LIN {X 0,Y 54.725,Z 1004.951,A -85,B 0,C 180,E1 26696.4,E2 26696.4} C_VEL
LIN {X 0,Y 49.29,Z 1006.172,A -85,B 0,C 180,E1 26729.997,E2 26729.997} C_VEL
LIN {X 0,Y 55.176,Z 1004.813,A -85,B 0,C 180,E1 26764.669,E2 26764.669} C_VEL
LIN {X 0,Y 77.211,Z 999.62,A -85,B 0,C 180,E1 26791.14,E2 26791.14} C_VEL
LIN {X 0,Y 112.41,Z 988.546,A -85,B 0,C 180,E1 26806.899,E2 26806.899} C_VEL
LIN {X 0,Y 149.803,Z 972.339,A -85,B 0,C 180,E1 26814.847,E2 26814.847} C_VEL
LIN {X 0,Y 181.716,Z 954.19,A -85,B 0,C 180,E1 26818.987,E2 26818.987} C_VEL
LIN {X 0,Y 144.346,Z 975.766,A -85,B 0,C 180,E1 26823.995,E2 26823.995} C_VEL
LIN {X 0,Y 128.492,Z 982.899,A -85,B 0,C 180,E1 26825.01,E2 26825.01} C_VEL
LIN {X 0,Y 112.377,Z 989.197,A -85,B 0,C 180,E1 26826.364,E2 26826.364} C_VEL
LIN {X 0,Y 79.371,Z 1000.218,A -85,B 0,C 180,E1 26837.491,E2 26837.491} C_VEL
LIN {X 0,Y 55.922,Z 1006.134,A -85,B 0,C 180,E1 26855.689,E2 26855.689} C_VEL
LIN {X 0,Y 42.006,Z 1009.143,A -85,B 0,C 180,E1 26888.877,E2 26888.877} C_VEL
LIN {X 0,Y 41.08,Z 1009.561,A -85,B 0,C 180,E1 26910.004,E2 26910.004} C_VEL
LIN {X 0,Y 47.227,Z 1008.017,A -85,B 0,C 180,E1 26949.886,E2 26949.886} C_VEL
LIN {X 0,Y 72.99,Z 1001.942,A -85,B 0,C 180,E1 26978.989,E2 26978.989} C_VEL
LIN {X 0,Y 110.548,Z 989.976,A -85,B 0,C 180,E1 26993.218,E2 26993.218} C_VEL
LIN {X 0,Y 149.583,Z 972.768,A -85,B 0,C 180,E1 26999.986,E2 26999.986} C_VEL
LIN {X 0,Y 157.146,Z 968.791,A -85,B 0,C 180,E1 27000.897,E2 27000.897} C_VEL
LIN {X 0,Y 117.393,Z 986.578,A -85,B 0,C 180,E1 27007.391,E2 27007.391} C_VEL
LIN {X 0,Y 80.336,Z 998.373,A -85,B 0,C 180,E1 27019.545,E2 27019.545} C_VEL
LIN {X 0,Y 57.052,Z 1003.65,A -85,B 0,C 180,E1 27037.231,E2 27037.231} C_VEL
LIN {X 0,Y 42.679,Z 1006.187,A -85,B 0,C 180,E1 27069.217,E2 27069.217} C_VEL
LIN {X 0,Y 41.362,Z 1006.47,A -85,B 0,C 180,E1 27089.996,E2 27089.996} C_VEL
LIN {X 0,Y 48.252,Z 1005.227,A -85,B 0,C 180,E1 27128.867,E2 27128.867} C_VEL
LIN {X 0,Y 74.683,Z 999.672,A -85,B 0,C 180,E1 27157.32,E2 27157.32} C_VEL
LIN {X 0,Y 107.56,Z 990.05,A -85,B 0,C 180,E1 27170.175,E2 27170.175} C_VEL
LIN {X 0,Y 148.509,Z 973.045,A -85,B 0,C 180,E1 27177.848,E2 27177.848} C_VEL
LIN {X 0,Y 157.303,Z 968.587,A -85,B 0,C 180,E1 27179.047,E2 27179.047} C_VEL
LIN {X 0,Y 117.818,Z 987.13,A -85,B 0,C 180,E1 27185.169,E2 27185.169} C_VEL
LIN {X 0,Y 112.377,Z 989.197,A -85,B 0,C 180,E1 27186.364,E2 27186.364} C_VEL
LIN {X 0,Y 96.022,Z 994.659,A -85,B 0,C 180,E1 27188.194,E2 27188.194} C_VEL
LIN {X 0,Y 79.547,Z 999.256,A -85,B 0,C 180,E1 27190.754,E2 27190.754} C_VEL
LIN {X 0,Y 51.572,Z 1005.826,A -85,B 0,C 180,E1 27208.272,E2 27208.272} C_VEL
LIN {X 0,Y 34.624,Z 1008.841,A -85,B 0,C 180,E1 27244.074,E2 27244.074} C_VEL
LIN {X 0,Y 33.124,Z 1009.263,A -85,B 0,C 180,E1 27270.005,E2 27270.005} C_VEL
LIN {X 0,Y 41.332,Z 1007.713,A -85,B 0,C 180,E1 27317.114,E2 27317.114} C_VEL
LIN {X 0,Y 70.453,Z 1001.634,A -85,B 0,C 180,E1 27345.266,E2 27345.266} C_VEL
LIN {X 0,Y 109.878,Z 989.667,A -85,B 0,C 180,E1 27357.503,E2 27357.503} C_VEL
LIN {X 0,Y 130.15,Z 981.612,A -85,B 0,C 180,E1 27361.203,E2 27361.203} C_VEL
LIN {X 0,Y 90.059,Z 995.489,A -85,B 0,C 180,E1 27369.654,E2 27369.654} C_VEL
LIN {X 0,Y 52.552,Z 1003.953,A -85,B 0,C 180,E1 27390.187,E2 27390.187} C_VEL
LIN {X 0,Y 35.329,Z 1006.487,A -85,B 0,C 180,E1 27424.618,E2 27424.618} C_VEL
LIN {X 0,Y 33.432,Z 1006.767,A -85,B 0,C 180,E1 27449.995,E2 27449.995} C_VEL
LIN {X 0,Y 42.315,Z 1005.527,A -85,B 0,C 180,E1 27495.689,E2 27495.689} C_VEL
LIN {X 0,Y 71.254,Z 1000.131,A -85,B 0,C 180,E1 27522.975,E2 27522.975} C_VEL
LIN {X 0,Y 106.472,Z 990.358,A -85,B 0,C 180,E1 27534.505,E2 27534.505} C_VEL
LIN {X 0,Y 130.541,Z 981.353,A -85,B 0,C 180,E1 27538.734,E2 27538.734} C_VEL
LIN {X 0,Y 97.059,Z 994.001,A -85,B 0,C 180,E1 27545.348,E2 27545.348} C_VEL
LIN {X 0,Y 79.547,Z 999.256,A -85,B 0,C 180,E1 27550.754,E2 27550.754} C_VEL
LIN {X 0,Y 63.154,Z 1003.048,A -85,B 0,C 180,E1 27554.617,E2 27554.617} C_VEL
LIN {X 0,Y 46.807,Z 1005.725,A -85,B 0,C 180,E1 27560.829,E2 27560.829} C_VEL
LIN {X 0,Y 27.615,Z 1008.539,A -85,B 0,C 180,E1 27596.758,E2 27596.758} C_VEL
LIN {X 0,Y 25.173,Z 1008.965,A -85,B 0,C 180,E1 27630.007,E2 27630.007} C_VEL
LIN {X 0,Y 36.292,Z 1007.408,A -85,B 0,C 180,E1 27686.561,E2 27686.561} C_VEL
LIN {X 0,Y 68.821,Z 1001.325,A -85,B 0,C 180,E1 27711.915,E2 27711.915} C_VEL
LIN {X 0,Y 98.808,Z 993.077,A -85,B 0,C 180,E1 27719.979,E2 27719.979} C_VEL
LIN {X 0,Y 103.722,Z 991.501,A -85,B 0,C 180,E1 27721.403,E2 27721.403} C_VEL
LIN {X 0,Y 60.756,Z 1002.242,A -85,B 0,C 180,E1 27734.393,E2 27734.393} C_VEL
LIN {X 0,Y 37.143,Z 1005.853,A -85,B 0,C 180,E1 27755.379,E2 27755.379} C_VEL
LIN {X 0,Y 25.522,Z 1007.064,A -85,B 0,C 180,E1 27809.994,E2 27809.994} C_VEL
LIN {X 0,Y 37.141,Z 1005.83,A -85,B 0,C 180,E1 27864.611,E2 27864.611} C_VEL
LIN {X 0,Y 69.31,Z 1000.437,A -85,B 0,C 180,E1 27889.418,E2 27889.418} C_VEL
LIN {X 0,Y 104.061,Z 991.318,A -85,B 0,C 180,E1 27898.558,E2 27898.558} C_VEL
LIN {X 0,Y 79.726,Z 998.59,A -85,B 0,C 180,E1 27904.443,E2 27904.443} C_VEL
LIN {X 0,Y 46.807,Z 1005.725,A -85,B 0,C 180,E1 27920.829,E2 27920.829} C_VEL
LIN {X 0,Y 31.263,Z 1007.541,A -85,B 0,C 180,E1 27932.406,E2 27932.406} C_VEL
LIN {X 0,Y 18.242,Z 1008.423,A -85,B 0,C 180,E1 27961.128,E2 27961.128} C_VEL
LIN {X 0,Y 17.205,Z 1008.666,A -85,B 0,C 180,E1 27990.01,E2 27990.01} C_VEL
LIN {X 0,Y 32.535,Z 1007.104,A -85,B 0,C 180,E1 28058.563,E2 28058.563} C_VEL
LIN {X 0,Y 72.688,Z 1000.024,A -85,B 0,C 180,E1 28079.971,E2 28079.971} C_VEL
LIN {X 0,Y 75.712,Z 999.346,A -85,B 0,C 180,E1 28080.652,E2 28080.652} C_VEL
LIN {X 0,Y 75.747,Z 999.286,A -85,B 0,C 180,E1 28081.86,E2 28081.86} C_VEL
LIN {X 0,Y 46.564,Z 1004.559,A -85,B 0,C 180,E1 28092.699,E2 28092.699} C_VEL
LIN {X 0,Y 21.994,Z 1007.085,A -85,B 0,C 180,E1 28126.485,E2 28126.485} C_VEL
LIN {X 0,Y 17.586,Z 1007.361,A -85,B 0,C 180,E1 28169.991,E2 28169.991} C_VEL
LIN {X 0,Y 33.143,Z 1006.131,A -85,B 0,C 180,E1 28236.005,E2 28236.005} C_VEL
LIN {X 0,Y 71.832,Z 1000.033,A -85,B 0,C 180,E1 28257.107,E2 28257.107} C_VEL
LIN {X 0,Y 75.745,Z 999.224,A -85,B 0,C 180,E1 28258.051,E2 28258.051} C_VEL
LIN {X 0,Y 75.707,Z 999.286,A -85,B 0,C 180,E1 28259.309,E2 28259.309} C_VEL
LIN {X 0,Y 42.748,Z 1005.659,A -85,B 0,C 180,E1 28272.114,E2 28272.114} C_VEL
LIN {X 0,Y 18.242,Z 1008.423,A -85,B 0,C 180,E1 28321.128,E2 28321.128} C_VEL
LIN {X 0,Y 13.954,Z 1008.54,A -85,B 0,C 180,E1 28348.35,E2 28348.35} C_VEL
LIN {X 0,Y 15.046,Z 1008,A -85,B 0,C 180,E1 28411.087,E2 28411.087} C_VEL
LIN {X 0,Y 45.426,Z 1004.937,A -85,B 0,C 180,E1 28440.165,E2 28440.165} C_VEL
LIN {X 0,Y 45.476,Z 1004.862,A -85,B 0,C 180,E1 28442.695,E2 28442.695} C_VEL
LIN {X 0,Y 17.115,Z 1007.384,A -85,B 0,C 180,E1 28467.769,E2 28467.769} C_VEL
LIN {X 0,Y 9.672,Z 1007.658,A -85,B 0,C 180,E1 28529.983,E2 28529.983} C_VEL
LIN {X 0,Y 30.76,Z 1006.434,A -85,B 0,C 180,E1 28609.855,E2 28609.855} C_VEL
LIN {X 0,Y 48.958,Z 1004.307,A -85,B 0,C 180,E1 28618.648,E2 28618.648} C_VEL
LIN {X 0,Y 16.67,Z 1007.934,A -85,B 0,C 180,E1 28644.759,E2 28644.759} C_VEL
LIN {X 0,Y 9.233,Z 1008.367,A -85,B 0,C 180,E1 28710.018,E2 28710.018} C_VEL
LIN {X 0,Y 15.046,Z 1008,A -85,B 0,C 180,E1 28771.087,E2 28771.087} C_VEL
LIN {X 0,Y 13.156,Z 1007.91,A -85,B 0,C 180,E1 28781.084,E2 28781.084} C_VEL
LIN {X 0,Y 3.411,Z 1007.913,A -85,B 0,C 180,E1 28817.533,E2 28817.533} C_VEL
LIN {X 0,Y 1.73,Z 1007.956,A -85,B 0,C 180,E1 28889.904,E2 28889.904} C_VEL
LIN {X 0,Y 8.337,Z 1007.838,A -85,B 0,C 180,E1 28980.252,E2 28980.252} C_VEL
LIN {X 0,Y 1.252,Z 1008.068,A -85,B 0,C 180,E1 29070.132,E2 29070.132} C_VEL
LIN {X 0,Y 8.174,Z 1007.847,A -85,B 0,C 180,E1 29159.743,E2 29159.743} C_VEL
LIN {X 0,Y 3.411,Z 1007.913,A -85,B 0,C 180,E1 29177.533,E2 29177.533} C_VEL
LIN {X 0,Y 1.959,Z 1009.913,A -85,B 0,C 180,E1 29207.521,E2 29207.521} C_VEL
LIN {X 0,Y 1.959,Z 1028,A -85,B 0,C 180,E1 29207.521,E2 29207.521} C_VEL
LIN {X 0,Y 1.959,Z 1028,A -85,B 0,C 180,E1 29207.521,E2 29207.521}

QRS_NEXT_CUT()
PTP {E1 29336.836,E2 29336.836}
PTP {X 0,Y 607.909,A -85,B 0,C 180,E1 29336.836,E2 29336.836,E3 0,E4 0,E5 0,E6 0}
QRS_SPEED_INIT()
LIN {X 0,Y 607.909,Z 1028,A -85,B 0,C 180,E1 29336.836,E2 29336.836,E3 0,E4 0,E5 0,E6 0} C_VEL
LIN {X 0,Y 607.909,Z 365.402,A -85,B 0,C 180,E1 29336.836,E2 29336.836} C_VEL
LIN {X 0,Y 607.909,Z 357.325,A -85,B 0,C 180,E1 29336.836,E2 29336.836} C_VEL
LIN {X 0,Y 607.881,Z 355.325,A -85,B 0,C 180,E1 29336.648,E2 29336.648} C_VEL
LIN {X 0,Y 607.838,Z 355.326,A -85,B 0,C 180,E1 29333.767,E2 29333.767} C_VEL
LIN {X 0,Y 607.91,Z 355.324,A -85,B 0,C 180,E1 29330.656,E2 29330.656} C_VEL
LIN {X 0,Y 607.845,Z 355.325,A -85,B 0,C 180,E1 29327.652,E2 29327.652} C_VEL
LIN {X 0,Y 607.919,Z 355.322,A -85,B 0,C 180,E1 29324.513,E2 29324.513} C_VEL
LIN {X 0,Y 607.851,Z 355.324,A -85,B 0,C 180,E1 29321.49,E2 29321.49} C_VEL
LIN {X 0,Y 607.914,Z 355.322,A -85,B 0,C 180,E1 29318.382,E2 29318.382} C_VEL
LIN {X 0,Y 607.857,Z 355.323,A -85,B 0,C 180,E1 29315.304,E2 29315.304} C_VEL
LIN {X 0,Y 607.917,Z 355.32,A -85,B 0,C 180,E1 29312.153,E2 29312.153} C_VEL
LIN {X 0,Y 607.865,Z 355.323,A -85,B 0,C 180,E1 29309.123,E2 29309.123} C_VEL
LIN {X 0,Y 607.915,Z 355.319,A -85,B 0,C 180,E1 29305.98,E2 29305.98} C_VEL
LIN {X 0,Y 607.873,Z 355.324,A -85,B 0,C 180,E1 29302.867,E2 29302.867} C_VEL
LIN {X 0,Y 607.914,Z 355.318,A -85,B 0,C 180,E1 29299.607,E2 29299.607} C_VEL
LIN {X 0,Y 607.902,Z 355.326,A -85,B 0,C 180,E1 29296.353,E2 29296.353} C_VEL
LIN {X 0,Y 607.886,Z 355.318,A -85,B 0,C 180,E1 29293.089,E2 29293.089} C_VEL
LIN {X 0,Y 607.913,Z 355.327,A -85,B 0,C 180,E1 29289.964,E2 29289.964} C_VEL
LIN {X 0,Y 607.907,Z 355.443,A -85,B 0,C 180,E1 29287.748,E2 29287.748} C_VEL
LIN {X 0,Y 607.908,Z 361.77,A -85,B 0,C 180,E1 29287.31,E2 29287.31} C_VEL
LIN {X 0,Y 607.919,Z 569.3,A -85,B 0,C 180,E1 29284.345,E2 29284.345} C_VEL
LIN {X 0,Y 607.911,Z 708.358,A -85,B 0,C 180,E1 29282.392,E2 29282.392} C_VEL
LIN {X 0,Y 607.914,Z 731.612,A -85,B 0,C 180,E1 29281.897,E2 29281.897} C_VEL
LIN {X 0,Y 607.916,Z 750.464,A -85,B 0,C 180,E1 29281.352,E2 29281.352} C_VEL
LIN {X 0,Y 607.912,Z 771.604,A -85,B 0,C 180,E1 29280.596,E2 29280.596} C_VEL
LIN {X 0,Y 607.917,Z 792.337,A -85,B 0,C 180,E1 29279.67,E2 29279.67} C_VEL
LIN {X 0,Y 607.916,Z 812.983,A -85,B 0,C 180,E1 29278.591,E2 29278.591} C_VEL
LIN {X 0,Y 607.917,Z 832.838,A -85,B 0,C 180,E1 29277.358,E2 29277.358} C_VEL
LIN {X 0,Y 607.912,Z 852.097,A -85,B 0,C 180,E1 29275.993,E2 29275.993} C_VEL
LIN {X 0,Y 607.909,Z 870.534,A -85,B 0,C 180,E1 29274.483,E2 29274.483} C_VEL
LIN {X 0,Y 607.916,Z 888.688,A -85,B 0,C 180,E1 29272.786,E2 29272.786} C_VEL
LIN {X 0,Y 607.914,Z 904.514,A -85,B 0,C 180,E1 29271.109,E2 29271.109} C_VEL
LIN {X 0,Y 607.913,Z 919.726,A -85,B 0,C 180,E1 29269.251,E2 29269.251} C_VEL
LIN {X 0,Y 607.913,Z 934.238,A -85,B 0,C 180,E1 29267.218,E2 29267.218} C_VEL
LIN {X 0,Y 607.896,Z 945.78,A -85,B 0,C 180,E1 29265.354,E2 29265.354} C_VEL
LIN {X 0,Y 607.887,Z 956.548,A -85,B 0,C 180,E1 29263.311,E2 29263.311} C_VEL
LIN {X 0,Y 607.91,Z 965.19,A -85,B 0,C 180,E1 29261.382,E2 29261.382} C_VEL
LIN {X 0,Y 607.892,Z 972.898,A -85,B 0,C 180,E1 29259.275,E2 29259.275} C_VEL
LIN {X 0,Y 607.89,Z 978.472,A -85,B 0,C 180,E1 29257.37,E2 29257.37} C_VEL
LIN {X 0,Y 607.909,Z 983.246,A -85,B 0,C 180,E1 29255.189,E2 29255.189} C_VEL
LIN {X 0,Y 607.882,Z 986.013,A -85,B 0,C 180,E1 29253.3,E2 29253.3} C_VEL
LIN {X 0,Y 607.909,Z 987.728,A -85,B 0,C 180,E1 29251.131,E2 29251.131} C_VEL
LIN {X 0,Y 607.883,Z 987.816,A -85,B 0,C 180,E1 29249.152,E2 29249.152} C_VEL
LIN {X 0,Y 607.886,Z 986.458,A -85,B 0,C 180,E1 29246.983,E2 29246.983} C_VEL
LIN {X 0,Y 607.904,Z 983.715,A -85,B 0,C 180,E1 29244.999,E2 29244.999} C_VEL
LIN {X 0,Y 607.88,Z 979.476,A -85,B 0,C 180,E1 29242.914,E2 29242.914} C_VEL
LIN {X 0,Y 607.914,Z 973.793,A -85,B 0,C 180,E1 29240.916,E2 29240.916} C_VEL
LIN {X 0,Y 607.889,Z 966.368,A -85,B 0,C 180,E1 29238.81,E2 29238.81} C_VEL
LIN {X 0,Y 607.89,Z 957.44,A -85,B 0,C 180,E1 29236.785,E2 29236.785} C_VEL
LIN {X 0,Y 607.911,Z 947.433,A -85,B 0,C 180,E1 29234.842,E2 29234.842} C_VEL
LIN {X 0,Y 607.904,Z 935.365,A -85,B 0,C 180,E1 29232.864,E2 29232.864} C_VEL
LIN {X 0,Y 607.903,Z 922.36,A -85,B 0,C 180,E1 29230.996,E2 29230.996} C_VEL
LIN {X 0,Y 607.913,Z 907.831,A -85,B 0,C 180,E1 29229.193,E2 29229.193} C_VEL
LIN {X 0,Y 607.915,Z 890.666,A -85,B 0,C 180,E1 29227.324,E2 29227.324} C_VEL
LIN {X 0,Y 607.905,Z 873.391,A -85,B 0,C 180,E1 29225.671,E2 29225.671} C_VEL
LIN {X 0,Y 607.908,Z 855.212,A -85,B 0,C 180,E1 29224.163,E2 29224.163} C_VEL
LIN {X 0,Y 607.914,Z 834.209,A -85,B 0,C 180,E1 29222.643,E2 29222.643} C_VEL
LIN {X 0,Y 607.917,Z 814.952,A -85,B 0,C 180,E1 29221.436,E2 29221.436} C_VEL
LIN {X 0,Y 607.918,Z 794.18,A -85,B 0,C 180,E1 29220.33,E2 29220.33} C_VEL
LIN {X 0,Y 607.914,Z 774.981,A -85,B 0,C 180,E1 29219.458,E2 29219.458} C_VEL
LIN {X 0,Y 607.913,Z 753.274,A -85,B 0,C 180,E1 29218.648,E2 29218.648} C_VEL
LIN {X 0,Y 607.911,Z 734.978,A -85,B 0,C 180,E1 29218.103,E2 29218.103} C_VEL
LIN {X 0,Y 607.912,Z 713.659,A -85,B 0,C 180,E1 29217.607,E2 29217.607} C_VEL
LIN {X 0,Y 607.916,Z 678.046,A -85,B 0,C 180,E1 29217.076,E2 29217.076} C_VEL
LIN {X 0,Y 607.907,Z 467.252,A -85,B 0,C 180,E1 29214.12,E2 29214.12} C_VEL
LIN {X 0,Y 607.908,Z 361.202,A -85,B 0,C 180,E1 29212.58,E2 29212.58} C_VEL
LIN {X 0,Y 607.905,Z 355.327,A -85,B 0,C 180,E1 29212.137,E2 29212.137} C_VEL
LIN {X 0,Y 607.891,Z 355.32,A -85,B 0,C 180,E1 29208.989,E2 29208.989} C_VEL
LIN {X 0,Y 607.916,Z 355.327,A -85,B 0,C 180,E1 29205.79,E2 29205.79} C_VEL
LIN {X 0,Y 607.907,Z 355.318,A -85,B 0,C 180,E1 29202.532,E2 29202.532} C_VEL
LIN {X 0,Y 607.887,Z 355.324,A -85,B 0,C 180,E1 29199.291,E2 29199.291} C_VEL
LIN {X 0,Y 607.915,Z 355.318,A -85,B 0,C 180,E1 29196.15,E2 29196.15} C_VEL
LIN {X 0,Y 607.874,Z 355.324,A -85,B 0,C 180,E1 29192.987,E2 29192.987} C_VEL
LIN {X 0,Y 607.915,Z 355.32,A -85,B 0,C 180,E1 29189.891,E2 29189.891} C_VEL
LIN {X 0,Y 607.866,Z 355.324,A -85,B 0,C 180,E1 29186.739,E2 29186.739} C_VEL
LIN {X 0,Y 607.916,Z 355.321,A -85,B 0,C 180,E1 29183.65,E2 29183.65} C_VEL
LIN {X 0,Y 607.858,Z 355.324,A -85,B 0,C 180,E1 29180.51,E2 29180.51} C_VEL
LIN {X 0,Y 607.917,Z 355.323,A -85,B 0,C 180,E1 29177.418,E2 29177.418} C_VEL
LIN {X 0,Y 607.851,Z 355.324,A -85,B 0,C 180,E1 29174.363,E2 29174.363} C_VEL
LIN {X 0,Y 607.918,Z 355.323,A -85,B 0,C 180,E1 29171.287,E2 29171.287} C_VEL
LIN {X 0,Y 607.845,Z 355.325,A -85,B 0,C 180,E1 29168.228,E2 29168.228} C_VEL
LIN {X 0,Y 607.911,Z 355.324,A -85,B 0,C 180,E1 29165.19,E2 29165.19} C_VEL
LIN {X 0,Y 607.837,Z 355.326,A -85,B 0,C 180,E1 29162.074,E2 29162.074} C_VEL
LIN {X 0,Y 607.89,Z 355.325,A -85,B 0,C 180,E1 29159.152,E2 29159.152} C_VEL
LIN {X 0,Y 607.832,Z 355.327,A -85,B 0,C 180,E1 29156.039,E2 29156.039} C_VEL
LIN {X 0,Y 607.846,Z 355.327,A -85,B 0,C 180,E1 29153.293,E2 29153.293} C_VEL
LIN {X 0,Y 607.837,Z 355.327,A -85,B 0,C 180,E1 29150.054,E2 29150.054} C_VEL
LIN {X 0,Y 607.833,Z 355.327,A -85,B 0,C 180,E1 29147.363,E2 29147.363} C_VEL
LIN {X 0,Y 607.874,Z 355.325,A -85,B 0,C 180,E1 29144.181,E2 29144.181} C_VEL
LIN {X 0,Y 607.837,Z 355.326,A -85,B 0,C 180,E1 29141.291,E2 29141.291} C_VEL
LIN {X 0,Y 607.904,Z 355.323,A -85,B 0,C 180,E1 29138.179,E2 29138.179} C_VEL
LIN {X 0,Y 607.842,Z 355.325,A -85,B 0,C 180,E1 29135.2,E2 29135.2} C_VEL
LIN {X 0,Y 607.919,Z 355.323,A -85,B 0,C 180,E1 29132.154,E2 29132.154} C_VEL
LIN {X 0,Y 607.85,Z 355.324,A -85,B 0,C 180,E1 29129.122,E2 29129.122} C_VEL
LIN {X 0,Y 607.918,Z 355.325,A -85,B 0,C 180,E1 29126.113,E2 29126.113} C_VEL
LIN {X 0,Y 607.857,Z 355.324,A -85,B 0,C 180,E1 29122.985,E2 29122.985} C_VEL
LIN {X 0,Y 607.915,Z 355.323,A -85,B 0,C 180,E1 29119.882,E2 29119.882} C_VEL
LIN {X 0,Y 607.863,Z 355.323,A -85,B 0,C 180,E1 29116.769,E2 29116.769} C_VEL
LIN {X 0,Y 607.913,Z 355.323,A -85,B 0,C 180,E1 29113.687,E2 29113.687} C_VEL
LIN {X 0,Y 607.869,Z 355.324,A -85,B 0,C 180,E1 29110.639,E2 29110.639} C_VEL
LIN {X 0,Y 607.914,Z 355.567,A -85,B 0,C 180,E1 29109.746,E2 29109.746} C_VEL
LIN {X 0,Y 607.913,Z 391.305,A -85,B 0,C 180,E1 29107.362,E2 29107.362} C_VEL
LIN {X 0,Y 607.916,Z 598.672,A -85,B 0,C 180,E1 29104.399,E2 29104.399} C_VEL
LIN {X 0,Y 607.913,Z 738.085,A -85,B 0,C 180,E1 29102.441,E2 29102.441} C_VEL
LIN {X 0,Y 607.915,Z 761.196,A -85,B 0,C 180,E1 29101.953,E2 29101.953} C_VEL
LIN {X 0,Y 607.916,Z 780.557,A -85,B 0,C 180,E1 29101.394,E2 29101.394} C_VEL
LIN {X 0,Y 607.911,Z 802.013,A -85,B 0,C 180,E1 29100.624,E2 29100.624} C_VEL
LIN {X 0,Y 607.919,Z 822.106,A -85,B 0,C 180,E1 29099.726,E2 29099.726} C_VEL
LIN {X 0,Y 607.916,Z 842.821,A -85,B 0,C 180,E1 29098.645,E2 29098.645} C_VEL
LIN {X 0,Y 607.916,Z 862.611,A -85,B 0,C 180,E1 29097.418,E2 29097.418} C_VEL
LIN {X 0,Y 607.912,Z 881.995,A -85,B 0,C 180,E1 29096.046,E2 29096.046} C_VEL
LIN {X 0,Y 607.91,Z 900.18,A -85,B 0,C 180,E1 29094.558,E2 29094.558} C_VEL
LIN {X 0,Y 607.916,Z 918.622,A -85,B 0,C 180,E1 29092.837,E2 29092.837} C_VEL
LIN {X 0,Y 607.91,Z 934.895,A -85,B 0,C 180,E1 29091.11,E2 29091.11} C_VEL
LIN {X 0,Y 607.91,Z 950.072,A -85,B 0,C 180,E1 29089.252,E2 29089.252} C_VEL
LIN {X 0,Y 607.911,Z 964.528,A -85,B 0,C 180,E1 29087.219,E2 29087.219} C_VEL
LIN {X 0,Y 607.9,Z 976.044,A -85,B 0,C 180,E1 29085.354,E2 29085.354} C_VEL
LIN {X 0,Y 607.886,Z 986.76,A -85,B 0,C 180,E1 29083.312,E2 29083.312} C_VEL
LIN {X 0,Y 607.907,Z 995.299,A -85,B 0,C 180,E1 29081.401,E2 29081.401} C_VEL
LIN {X 0,Y 607.896,Z 1003.04,A -85,B 0,C 180,E1 29079.275,E2 29079.275} C_VEL
LIN {X 0,Y 607.888,Z 1008.591,A -85,B 0,C 180,E1 29077.37,E2 29077.37} C_VEL
LIN {X 0,Y 607.911,Z 1013.32,A -85,B 0,C 180,E1 29075.19,E2 29075.19} C_VEL
LIN {X 0,Y 607.881,Z 1016.139,A -85,B 0,C 180,E1 29073.239,E2 29073.239} C_VEL
LIN {X 0,Y 607.897,Z 1017.761,A -85,B 0,C 180,E1 29071.037,E2 29071.037} C_VEL
LIN {X 0,Y 607.886,Z 1017.806,A -85,B 0,C 180,E1 29069.152,E2 29069.152} C_VEL
LIN {X 0,Y 607.884,Z 1016.405,A -85,B 0,C 180,E1 29066.984,E2 29066.984} C_VEL
LIN {X 0,Y 607.907,Z 1013.64,A -85,B 0,C 180,E1 29065,E2 29065} C_VEL
LIN {X 0,Y 607.882,Z 1009.103,A -85,B 0,C 180,E1 29062.82,E2 29062.82} C_VEL
LIN {X 0,Y 607.904,Z 1003.346,A -85,B 0,C 180,E1 29060.821,E2 29060.821} C_VEL
LIN {X 0,Y 607.898,Z 995.791,A -85,B 0,C 180,E1 29058.714,E2 29058.714} C_VEL
LIN {X 0,Y 607.888,Z 987.227,A -85,B 0,C 180,E1 29056.786,E2 29056.786} C_VEL
LIN {X 0,Y 607.911,Z 977.193,A -85,B 0,C 180,E1 29054.842,E2 29054.842} C_VEL
LIN {X 0,Y 607.908,Z 965.052,A -85,B 0,C 180,E1 29052.861,E2 29052.861} C_VEL
LIN {X 0,Y 607.906,Z 951.236,A -85,B 0,C 180,E1 29050.897,E2 29050.897} C_VEL
LIN {X 0,Y 607.91,Z 936.603,A -85,B 0,C 180,E1 29049.092,E2 29049.092} C_VEL
LIN {X 0,Y 607.914,Z 920.209,A -85,B 0,C 180,E1 29047.323,E2 29047.323} C_VEL
LIN {X 0,Y 607.905,Z 902.853,A -85,B 0,C 180,E1 29045.67,E2 29045.67} C_VEL
LIN {X 0,Y 607.908,Z 884.65,A -85,B 0,C 180,E1 29044.164,E2 29044.164} C_VEL
LIN {X 0,Y 607.913,Z 864.224,A -85,B 0,C 180,E1 29042.689,E2 29042.689} C_VEL
LIN {X 0,Y 607.916,Z 844.862,A -85,B 0,C 180,E1 29041.476,E2 29041.476} C_VEL
LIN {X 0,Y 607.918,Z 824.383,A -85,B 0,C 180,E1 29040.384,E2 29040.384} C_VEL
LIN {X 0,Y 607.914,Z 805.451,A -85,B 0,C 180,E1 29039.523,E2 29039.523} C_VEL
LIN {X 0,Y 607.914,Z 783.164,A -85,B 0,C 180,E1 29038.69,E2 29038.69} C_VEL
LIN {X 0,Y 607.913,Z 764.563,A -85,B 0,C 180,E1 29038.137,E2 29038.137} C_VEL
LIN {X 0,Y 607.912,Z 742.819,A -85,B 0,C 180,E1 29037.636,E2 29037.636} C_VEL
LIN {X 0,Y 607.915,Z 700.755,A -85,B 0,C 180,E1 29037.02,E2 29037.02} C_VEL
LIN {X 0,Y 607.904,Z 492.11,A -85,B 0,C 180,E1 29034.092,E2 29034.092} C_VEL
LIN {X 0,Y 607.913,Z 390.704,A -85,B 0,C 180,E1 29032.619,E2 29032.619} C_VEL
LIN {X 0,Y 607.914,Z 355.327,A -85,B 0,C 180,E1 29030.229,E2 29030.229} C_VEL
LIN {X 0,Y 607.867,Z 355.323,A -85,B 0,C 180,E1 29027.189,E2 29027.189} C_VEL
LIN {X 0,Y 607.917,Z 355.326,A -85,B 0,C 180,E1 29024.056,E2 29024.056} C_VEL
LIN {X 0,Y 607.864,Z 355.323,A -85,B 0,C 180,E1 29020.983,E2 29020.983} C_VEL
LIN {X 0,Y 607.913,Z 355.328,A -85,B 0,C 180,E1 29017.842,E2 29017.842} C_VEL
LIN {X 0,Y 607.857,Z 355.323,A -85,B 0,C 180,E1 29014.804,E2 29014.804} C_VEL
LIN {X 0,Y 607.908,Z 355.327,A -85,B 0,C 180,E1 29011.646,E2 29011.646} C_VEL
LIN {X 0,Y 607.849,Z 355.323,A -85,B 0,C 180,E1 29008.706,E2 29008.706} C_VEL
LIN {X 0,Y 607.919,Z 355.327,A -85,B 0,C 180,E1 29005.63,E2 29005.63} C_VEL
LIN {X 0,Y 607.841,Z 355.325,A -85,B 0,C 180,E1 29002.638,E2 29002.638} C_VEL
LIN {X 0,Y 607.916,Z 355.326,A -85,B 0,C 180,E1 28999.556,E2 28999.556} C_VEL
LIN {X 0,Y 607.835,Z 355.326,A -85,B 0,C 180,E1 28996.533,E2 28996.533} C_VEL
LIN {X 0,Y 607.894,Z 355.326,A -85,B 0,C 180,E1 28993.602,E2 28993.602} C_VEL
LIN {X 0,Y 607.831,Z 355.327,A -85,B 0,C 180,E1 28990.52,E2 28990.52} C_VEL
LIN {X 0,Y 607.857,Z 355.327,A -85,B 0,C 180,E1 28987.656,E2 28987.656} C_VEL
LIN {X 0,Y 607.837,Z 355.327,A -85,B 0,C 180,E1 28984.528,E2 28984.528} C_VEL
LIN {X 0,Y 607.836,Z 355.327,A -85,B 0,C 180,E1 28981.791,E2 28981.791} C_VEL
LIN {X 0,Y 607.865,Z 355.325,A -85,B 0,C 180,E1 28978.586,E2 28978.586} C_VEL
LIN {X 0,Y 607.881,Z 355.325,A -85,B 0,C 180,E1 28976.648,E2 28976.648} C_VEL
LIN {X 0,Y 606.822,Z 355.456,A -85,B 0,C 180,E1 28975.922,E2 28975.922} C_VEL
LIN {X 0,Y 600.411,Z 356.253,A -85,B 0,C 180,E1 28973.885,E2 28973.885} C_VEL
LIN {X 0,Y 599.924,Z 356.316,A -85,B 0,C 180,E1 28973.355,E2 28973.355} C_VEL
LIN {X 0,Y 599.914,Z 356.314,A -85,B 0,C 180,E1 28970.115,E2 28970.115} C_VEL
LIN {X 0,Y 599.922,Z 356.315,A -85,B 0,C 180,E1 28967.291,E2 28967.291} C_VEL
LIN {X 0,Y 599.927,Z 356.311,A -85,B 0,C 180,E1 28964.038,E2 28964.038} C_VEL
LIN {X 0,Y 599.928,Z 356.313,A -85,B 0,C 180,E1 28961.136,E2 28961.136} C_VEL
LIN {X 0,Y 599.934,Z 356.31,A -85,B 0,C 180,E1 28957.873,E2 28957.873} C_VEL
LIN {X 0,Y 599.945,Z 356.313,A -85,B 0,C 180,E1 28954.851,E2 28954.851} C_VEL
LIN {X 0,Y 599.934,Z 356.31,A -85,B 0,C 180,E1 28951.626,E2 28951.626} C_VEL
LIN {X 0,Y 599.965,Z 356.315,A -85,B 0,C 180,E1 28948.557,E2 28948.557} C_VEL
LIN {X 0,Y 599.933,Z 356.308,A -85,B 0,C 180,E1 28945.367,E2 28945.367} C_VEL
LIN {X 0,Y 599.978,Z 356.315,A -85,B 0,C 180,E1 28942.294,E2 28942.294} C_VEL
LIN {X 0,Y 599.936,Z 356.311,A -85,B 0,C 180,E1 28939.082,E2 28939.082} C_VEL
LIN {X 0,Y 599.971,Z 356.313,A -85,B 0,C 180,E1 28935.904,E2 28935.904} C_VEL
LIN {X 0,Y 599.939,Z 356.308,A -85,B 0,C 180,E1 28932.835,E2 28932.835} C_VEL
LIN {X 0,Y 599.97,Z 356.315,A -85,B 0,C 180,E1 28929.782,E2 28929.782} C_VEL
LIN {X 0,Y 599.967,Z 356.378,A -85,B 0,C 180,E1 28928.269,E2 28928.269} C_VEL
LIN {X 0,Y 601.089,Z 359.961,A -85,B 0,C 180,E1 28927.92,E2 28927.92} C_VEL
LIN {X 0,Y 601.275,Z 362.256,A -85,B 0,C 180,E1 28927.787,E2 28927.787} C_VEL
LIN {X 0,Y 601.536,Z 366.664,A -85,B 0,C 180,E1 28927.702,E2 28927.702} C_VEL
LIN {X 0,Y 601.303,Z 574.213,A -85,B 0,C 180,E1 28924.708,E2 28924.708} C_VEL
LIN {X 0,Y 601.145,Z 709.258,A -85,B 0,C 180,E1 28922.788,E2 28922.788} C_VEL
LIN {X 0,Y 601.066,Z 733.04,A -85,B 0,C 180,E1 28922.266,E2 28922.266} C_VEL
LIN {X 0,Y 601,Z 752.537,A -85,B 0,C 180,E1 28921.688,E2 28921.688} C_VEL
LIN {X 0,Y 600.875,Z 775.465,A -85,B 0,C 180,E1 28920.827,E2 28920.827} C_VEL
LIN {X 0,Y 600.791,Z 794.591,A -85,B 0,C 180,E1 28919.948,E2 28919.948} C_VEL
LIN {X 0,Y 600.649,Z 816.578,A -85,B 0,C 180,E1 28918.752,E2 28918.752} C_VEL
LIN {X 0,Y 600.552,Z 835.962,A -85,B 0,C 180,E1 28917.513,E2 28917.513} C_VEL
LIN {X 0,Y 600.414,Z 856.076,A -85,B 0,C 180,E1 28916.024,E2 28916.024} C_VEL
LIN {X 0,Y 600.306,Z 874.696,A -85,B 0,C 180,E1 28914.447,E2 28914.447} C_VEL
LIN {X 0,Y 600.224,Z 891.736,A -85,B 0,C 180,E1 28912.784,E2 28912.784} C_VEL
LIN {X 0,Y 600.132,Z 907.933,A -85,B 0,C 180,E1 28910.987,E2 28910.987} C_VEL
LIN {X 0,Y 600.07,Z 922.642,A -85,B 0,C 180,E1 28909.134,E2 28909.134} C_VEL
LIN {X 0,Y 600.012,Z 936.173,A -85,B 0,C 180,E1 28907.152,E2 28907.152} C_VEL
LIN {X 0,Y 599.975,Z 948.523,A -85,B 0,C 180,E1 28905.066,E2 28905.066} C_VEL
LIN {X 0,Y 599.926,Z 957.943,A -85,B 0,C 180,E1 28903.197,E2 28903.197} C_VEL
LIN {X 0,Y 599.911,Z 966.752,A -85,B 0,C 180,E1 28901.146,E2 28901.146} C_VEL
LIN {X 0,Y 599.914,Z 973.815,A -85,B 0,C 180,E1 28899.109,E2 28899.109} C_VEL
LIN {X 0,Y 599.884,Z 979.713,A -85,B 0,C 180,E1 28896.988,E2 28896.988} C_VEL
LIN {X 0,Y 599.904,Z 983.883,A -85,B 0,C 180,E1 28894.875,E2 28894.875} C_VEL
LIN {X 0,Y 599.896,Z 986.682,A -85,B 0,C 180,E1 28892.77,E2 28892.77} C_VEL
LIN {X 0,Y 599.885,Z 987.84,A -85,B 0,C 180,E1 28890.668,E2 28890.668} C_VEL
LIN {X 0,Y 599.913,Z 987.679,A -85,B 0,C 180,E1 28888.567,E2 28888.567} C_VEL
LIN {X 0,Y 599.888,Z 985.894,A -85,B 0,C 180,E1 28886.465,E2 28886.465} C_VEL
LIN {X 0,Y 599.9,Z 982.918,A -85,B 0,C 180,E1 28884.453,E2 28884.453} C_VEL
LIN {X 0,Y 599.917,Z 977.946,A -85,B 0,C 180,E1 28882.242,E2 28882.242} C_VEL
LIN {X 0,Y 599.893,Z 971.963,A -85,B 0,C 180,E1 28880.213,E2 28880.213} C_VEL
LIN {X 0,Y 599.929,Z 963.811,A -85,B 0,C 180,E1 28878.045,E2 28878.045} C_VEL
LIN {X 0,Y 599.957,Z 954.654,A -85,B 0,C 180,E1 28876.017,E2 28876.017} C_VEL
LIN {X 0,Y 599.969,Z 943.986,A -85,B 0,C 180,E1 28874.041,E2 28874.041} C_VEL
LIN {X 0,Y 600.019,Z 931.599,A -85,B 0,C 180,E1 28872.046,E2 28872.046} C_VEL
LIN {X 0,Y 600.075,Z 917.688,A -85,B 0,C 180,E1 28870.131,E2 28870.131} C_VEL
LIN {X 0,Y 600.16,Z 901.624,A -85,B 0,C 180,E1 28868.193,E2 28868.193} C_VEL
LIN {X 0,Y 600.254,Z 885.004,A -85,B 0,C 180,E1 28866.439,E2 28866.439} C_VEL
LIN {X 0,Y 600.349,Z 867.341,A -85,B 0,C 180,E1 28864.819,E2 28864.819} C_VEL
LIN {X 0,Y 600.476,Z 847.548,A -85,B 0,C 180,E1 28863.228,E2 28863.228} C_VEL
LIN {X 0,Y 600.576,Z 828.468,A -85,B 0,C 180,E1 28861.894,E2 28861.894} C_VEL
LIN {X 0,Y 600.716,Z 807.691,A -85,B 0,C 180,E1 28860.651,E2 28860.651} C_VEL
LIN {X 0,Y 600.81,Z 787.451,A -85,B 0,C 180,E1 28859.612,E2 28859.612} C_VEL
LIN {X 0,Y 600.94,Z 765.942,A -85,B 0,C 180,E1 28858.703,E2 28858.703} C_VEL
LIN {X 0,Y 601.012,Z 746.205,A -85,B 0,C 180,E1 28858.017,E2 28858.017} C_VEL
LIN {X 0,Y 601.11,Z 723.027,A -85,B 0,C 180,E1 28857.4,E2 28857.4} C_VEL
LIN {X 0,Y 601.155,Z 703.845,A -85,B 0,C 180,E1 28857.033,E2 28857.033} C_VEL
LIN {X 0,Y 601.392,Z 482.167,A -85,B 0,C 180,E1 28853.887,E2 28853.887} C_VEL
LIN {X 0,Y 601.358,Z 362.629,A -85,B 0,C 180,E1 28852.135,E2 28852.135} C_VEL
LIN {X 0,Y 601.083,Z 360.672,A -85,B 0,C 180,E1 28852.042,E2 28852.042} C_VEL
LIN {X 0,Y 600.876,Z 359.126,A -85,B 0,C 180,E1 28851.913,E2 28851.913} C_VEL
LIN {X 0,Y 599.958,Z 356.317,A -85,B 0,C 180,E1 28851.631,E2 28851.631} C_VEL
LIN {X 0,Y 599.971,Z 356.309,A -85,B 0,C 180,E1 28848.44,E2 28848.44} C_VEL
LIN {X 0,Y 599.944,Z 356.313,A -85,B 0,C 180,E1 28845.232,E2 28845.232} C_VEL
LIN {X 0,Y 599.97,Z 356.311,A -85,B 0,C 180,E1 28842.062,E2 28842.062} C_VEL
LIN {X 0,Y 599.938,Z 356.309,A -85,B 0,C 180,E1 28838.902,E2 28838.902} C_VEL
LIN {X 0,Y 599.976,Z 356.315,A -85,B 0,C 180,E1 28835.681,E2 28835.681} C_VEL
LIN {X 0,Y 599.94,Z 356.31,A -85,B 0,C 180,E1 28832.52,E2 28832.52} C_VEL
LIN {X 0,Y 599.955,Z 356.314,A -85,B 0,C 180,E1 28829.229,E2 28829.229} C_VEL
LIN {X 0,Y 599.954,Z 356.309,A -85,B 0,C 180,E1 28826.081,E2 28826.081} C_VEL
LIN {X 0,Y 599.93,Z 356.313,A -85,B 0,C 180,E1 28822.847,E2 28822.847} C_VEL
LIN {X 0,Y 599.963,Z 356.31,A -85,B 0,C 180,E1 28819.774,E2 28819.774} C_VEL
LIN {X 0,Y 599.921,Z 356.312,A -85,B 0,C 180,E1 28816.621,E2 28816.621} C_VEL
LIN {X 0,Y 599.96,Z 356.311,A -85,B 0,C 180,E1 28813.591,E2 28813.591} C_VEL
LIN {X 0,Y 599.915,Z 356.315,A -85,B 0,C 180,E1 28810.467,E2 28810.467} C_VEL
LIN {X 0,Y 599.936,Z 356.312,A -85,B 0,C 180,E1 28807.566,E2 28807.566} C_VEL
LIN {X 0,Y 599.912,Z 356.315,A -85,B 0,C 180,E1 28804.397,E2 28804.397} C_VEL
LIN {X 0,Y 599.917,Z 356.314,A -85,B 0,C 180,E1 28801.528,E2 28801.528} C_VEL
LIN {X 0,Y 599.908,Z 356.315,A -85,B 0,C 180,E1 28798.281,E2 28798.281} C_VEL
LIN {X 0,Y 599.899,Z 356.316,A -85,B 0,C 180,E1 28795.507,E2 28795.507} C_VEL
LIN {X 0,Y 599.91,Z 356.316,A -85,B 0,C 180,E1 28792.242,E2 28792.242} C_VEL
LIN {X 0,Y 599.891,Z 356.316,A -85,B 0,C 180,E1 28789.436,E2 28789.436} C_VEL
LIN {X 0,Y 599.94,Z 356.315,A -85,B 0,C 180,E1 28786.293,E2 28786.293} C_VEL
LIN {X 0,Y 599.895,Z 356.315,A -85,B 0,C 180,E1 28783.387,E2 28783.387} C_VEL
LIN {X 0,Y 599.967,Z 356.314,A -85,B 0,C 180,E1 28780.302,E2 28780.302} C_VEL
LIN {X 0,Y 599.901,Z 356.314,A -85,B 0,C 180,E1 28777.356,E2 28777.356} C_VEL
LIN {X 0,Y 599.98,Z 356.316,A -85,B 0,C 180,E1 28774.324,E2 28774.324} C_VEL
LIN {X 0,Y 599.909,Z 356.312,A -85,B 0,C 180,E1 28771.206,E2 28771.206} C_VEL
LIN {X 0,Y 599.975,Z 356.315,A -85,B 0,C 180,E1 28768.192,E2 28768.192} C_VEL
LIN {X 0,Y 599.916,Z 356.312,A -85,B 0,C 180,E1 28765.017,E2 28765.017} C_VEL
LIN {X 0,Y 599.977,Z 356.312,A -85,B 0,C 180,E1 28761.932,E2 28761.932} C_VEL
LIN {X 0,Y 599.921,Z 356.313,A -85,B 0,C 180,E1 28758.828,E2 28758.828} C_VEL
LIN {X 0,Y 599.977,Z 356.31,A -85,B 0,C 180,E1 28755.631,E2 28755.631} C_VEL
LIN {X 0,Y 599.93,Z 356.315,A -85,B 0,C 180,E1 28752.554,E2 28752.554} C_VEL
LIN {X 0,Y 599.956,Z 356.435,A -85,B 0,C 180,E1 28750.321,E2 28750.321} C_VEL
LIN {X 0,Y 601.277,Z 360.206,A -85,B 0,C 180,E1 28749.952,E2 28749.952} C_VEL
LIN {X 0,Y 601.27,Z 391.507,A -85,B 0,C 180,E1 28747.843,E2 28747.843} C_VEL
LIN {X 0,Y 601.541,Z 396.126,A -85,B 0,C 180,E1 28747.755,E2 28747.755} C_VEL
LIN {X 0,Y 601.3,Z 606.057,A -85,B 0,C 180,E1 28744.727,E2 28744.727} C_VEL
LIN {X 0,Y 601.147,Z 739.177,A -85,B 0,C 180,E1 28742.834,E2 28742.834} C_VEL
LIN {X 0,Y 601.066,Z 762.936,A -85,B 0,C 180,E1 28742.314,E2 28742.314} C_VEL
LIN {X 0,Y 601,Z 782.42,A -85,B 0,C 180,E1 28741.736,E2 28741.736} C_VEL
LIN {X 0,Y 600.875,Z 805.337,A -85,B 0,C 180,E1 28740.878,E2 28740.878} C_VEL
LIN {X 0,Y 600.793,Z 824.374,A -85,B 0,C 180,E1 28740.003,E2 28740.003} C_VEL
LIN {X 0,Y 600.65,Z 846.414,A -85,B 0,C 180,E1 28738.807,E2 28738.807} C_VEL
LIN {X 0,Y 600.552,Z 865.823,A -85,B 0,C 180,E1 28737.568,E2 28737.568} C_VEL
LIN {X 0,Y 600.413,Z 885.969,A -85,B 0,C 180,E1 28736.078,E2 28736.078} C_VEL
LIN {X 0,Y 600.308,Z 904.611,A -85,B 0,C 180,E1 28734.499,E2 28734.499} C_VEL
LIN {X 0,Y 600.225,Z 921.664,A -85,B 0,C 180,E1 28732.836,E2 28732.836} C_VEL
LIN {X 0,Y 600.128,Z 938.303,A -85,B 0,C 180,E1 28730.988,E2 28730.988} C_VEL
LIN {X 0,Y 600.066,Z 952.978,A -85,B 0,C 180,E1 28729.134,E2 28729.134} C_VEL
LIN {X 0,Y 600.009,Z 966.459,A -85,B 0,C 180,E1 28727.153,E2 28727.153} C_VEL
LIN {X 0,Y 599.973,Z 978.757,A -85,B 0,C 180,E1 28725.067,E2 28725.067} C_VEL
LIN {X 0,Y 599.926,Z 988.153,A -85,B 0,C 180,E1 28723.197,E2 28723.197} C_VEL
LIN {X 0,Y 599.905,Z 997.271,A -85,B 0,C 180,E1 28721.049,E2 28721.049} C_VEL
LIN {X 0,Y 599.92,Z 1003.955,A -85,B 0,C 180,E1 28719.109,E2 28719.109} C_VEL
LIN {X 0,Y 599.885,Z 1009.808,A -85,B 0,C 180,E1 28716.988,E2 28716.988} C_VEL
LIN {X 0,Y 599.906,Z 1013.798,A -85,B 0,C 180,E1 28714.972,E2 28714.972} C_VEL
LIN {X 0,Y 599.892,Z 1016.63,A -85,B 0,C 180,E1 28712.866,E2 28712.866} C_VEL
LIN {X 0,Y 599.883,Z 1017.828,A -85,B 0,C 180,E1 28710.764,E2 28710.764} C_VEL
LIN {X 0,Y 599.915,Z 1017.694,A -85,B 0,C 180,E1 28708.663,E2 28708.663} C_VEL
LIN {X 0,Y 599.886,Z 1015.954,A -85,B 0,C 180,E1 28706.561,E2 28706.561} C_VEL
LIN {X 0,Y 599.9,Z 1013.003,A -85,B 0,C 180,E1 28704.549,E2 28704.549} C_VEL
LIN {X 0,Y 599.914,Z 1008.083,A -85,B 0,C 180,E1 28702.339,E2 28702.339} C_VEL
LIN {X 0,Y 599.893,Z 1002.432,A -85,B 0,C 180,E1 28700.407,E2 28700.407} C_VEL
LIN {X 0,Y 599.929,Z 994.156,A -85,B 0,C 180,E1 28698.172,E2 28698.172} C_VEL
LIN {X 0,Y 599.935,Z 985.837,A -85,B 0,C 180,E1 28696.312,E2 28696.312} C_VEL
LIN {X 0,Y 599.967,Z 974.307,A -85,B 0,C 180,E1 28694.141,E2 28694.141} C_VEL
LIN {X 0,Y 600.009,Z 962.605,A -85,B 0,C 180,E1 28692.247,E2 28692.247} C_VEL
LIN {X 0,Y 600.08,Z 948.549,A -85,B 0,C 180,E1 28690.288,E2 28690.288} C_VEL
LIN {X 0,Y 600.163,Z 933.082,A -85,B 0,C 180,E1 28688.399,E2 28688.399} C_VEL
LIN {X 0,Y 600.237,Z 917.106,A -85,B 0,C 180,E1 28686.698,E2 28686.698} C_VEL
LIN {X 0,Y 600.347,Z 899.248,A -85,B 0,C 180,E1 28685.03,E2 28685.03} C_VEL
LIN {X 0,Y 600.47,Z 880.647,A -85,B 0,C 180,E1 28683.5,E2 28683.5} C_VEL
LIN {X 0,Y 600.566,Z 861.017,A -85,B 0,C 180,E1 28682.111,E2 28682.111} C_VEL
LIN {X 0,Y 600.708,Z 839.865,A -85,B 0,C 180,E1 28680.815,E2 28680.815} C_VEL
LIN {X 0,Y 600.801,Z 819.802,A -85,B 0,C 180,E1 28679.772,E2 28679.772} C_VEL
LIN {X 0,Y 600.931,Z 797.651,A -85,B 0,C 180,E1 28678.812,E2 28678.812} C_VEL
LIN {X 0,Y 601.009,Z 777.892,A -85,B 0,C 180,E1 28678.117,E2 28678.117} C_VEL
LIN {X 0,Y 601.108,Z 754.847,A -85,B 0,C 180,E1 28677.485,E2 28677.485} C_VEL
LIN {X 0,Y 601.153,Z 735.128,A -85,B 0,C 180,E1 28677.099,E2 28677.099} C_VEL
LIN {X 0,Y 601.389,Z 512.223,A -85,B 0,C 180,E1 28673.932,E2 28673.932} C_VEL
LIN {X 0,Y 601.372,Z 391.988,A -85,B 0,C 180,E1 28672.171,E2 28672.171} C_VEL
LIN {X 0,Y 601.151,Z 390.112,A -85,B 0,C 180,E1 28672.085,E2 28672.085} C_VEL
LIN {X 0,Y 601.121,Z 359.571,A -85,B 0,C 180,E1 28669.992,E2 28669.992} C_VEL
LIN {X 0,Y 599.939,Z 356.317,A -85,B 0,C 180,E1 28669.657,E2 28669.657} C_VEL
LIN {X 0,Y 599.978,Z 356.31,A -85,B 0,C 180,E1 28666.514,E2 28666.514} C_VEL
LIN {X 0,Y 599.928,Z 356.313,A -85,B 0,C 180,E1 28663.365,E2 28663.365} C_VEL
LIN {X 0,Y 599.979,Z 356.31,A -85,B 0,C 180,E1 28660.256,E2 28660.256} C_VEL
LIN {X 0,Y 599.92,Z 356.314,A -85,B 0,C 180,E1 28657.108,E2 28657.108} C_VEL
LIN {X 0,Y 599.979,Z 356.31,A -85,B 0,C 180,E1 28654.051,E2 28654.051} C_VEL
LIN {X 0,Y 599.914,Z 356.314,A -85,B 0,C 180,E1 28650.997,E2 28650.997} C_VEL
LIN {X 0,Y 599.977,Z 356.309,A -85,B 0,C 180,E1 28647.923,E2 28647.923} C_VEL
LIN {X 0,Y 599.906,Z 356.313,A -85,B 0,C 180,E1 28644.835,E2 28644.835} C_VEL
LIN {X 0,Y 599.96,Z 356.311,A -85,B 0,C 180,E1 28641.852,E2 28641.852} C_VEL
LIN {X 0,Y 599.903,Z 356.313,A -85,B 0,C 180,E1 28638.764,E2 28638.764} C_VEL
LIN {X 0,Y 599.922,Z 356.313,A -85,B 0,C 180,E1 28635.942,E2 28635.942} C_VEL
LIN {X 0,Y 599.902,Z 356.315,A -85,B 0,C 180,E1 28632.709,E2 28632.709} C_VEL
LIN {X 0,Y 599.899,Z 356.316,A -85,B 0,C 180,E1 28629.967,E2 28629.967} C_VEL
LIN {X 0,Y 599.899,Z 356.316,A -85,B 0,C 180,E1 28626.604,E2 28626.604} C_VEL
LIN {X 0,Y 599.896,Z 356.317,A -85,B 0,C 180,E1 28623.822,E2 28623.822} C_VEL
LIN {X 0,Y 599.917,Z 356.315,A -85,B 0,C 180,E1 28620.573,E2 28620.573} C_VEL
LIN {X 0,Y 599.896,Z 356.315,A -85,B 0,C 180,E1 28617.803,E2 28617.803} C_VEL
LIN {X 0,Y 599.952,Z 356.313,A -85,B 0,C 180,E1 28614.645,E2 28614.645} C_VEL
LIN {X 0,Y 599.924,Z 356.316,A -85,B 0,C 180,E1 28613.355,E2 28613.355} C_VEL
LIN {X 0,Y 598.984,Z 356.44,A -85,B 0,C 180,E1 28612.619,E2 28612.619} C_VEL
LIN {X 0,Y 592.429,Z 357.251,A -85,B 0,C 180,E1 28610.502,E2 28610.502} C_VEL
LIN {X 0,Y 591.97,Z 357.303,A -85,B 0,C 180,E1 28610.018,E2 28610.018} C_VEL
LIN {X 0,Y 591.999,Z 357.304,A -85,B 0,C 180,E1 28607.118,E2 28607.118} C_VEL
LIN {X 0,Y 591.98,Z 357.299,A -85,B 0,C 180,E1 28603.919,E2 28603.919} C_VEL
LIN {X 0,Y 592.015,Z 357.302,A -85,B 0,C 180,E1 28600.874,E2 28600.874} C_VEL
LIN {X 0,Y 591.983,Z 357.3,A -85,B 0,C 180,E1 28597.665,E2 28597.665} C_VEL
LIN {X 0,Y 592.032,Z 357.302,A -85,B 0,C 180,E1 28594.598,E2 28594.598} C_VEL
LIN {X 0,Y 591.986,Z 357.299,A -85,B 0,C 180,E1 28591.422,E2 28591.422} C_VEL
LIN {X 0,Y 592.038,Z 357.304,A -85,B 0,C 180,E1 28588.316,E2 28588.316} C_VEL
LIN {X 0,Y 591.989,Z 357.297,A -85,B 0,C 180,E1 28585.159,E2 28585.159} C_VEL
LIN {X 0,Y 592.035,Z 357.299,A -85,B 0,C 180,E1 28582.055,E2 28582.055} C_VEL
LIN {X 0,Y 591.997,Z 357.302,A -85,B 0,C 180,E1 28578.867,E2 28578.867} C_VEL
LIN {X 0,Y 592.039,Z 357.297,A -85,B 0,C 180,E1 28575.585,E2 28575.585} C_VEL
LIN {X 0,Y 592.023,Z 357.299,A -85,B 0,C 180,E1 28572.291,E2 28572.291} C_VEL
LIN {X 0,Y 592.017,Z 357.301,A -85,B 0,C 180,E1 28569.023,E2 28569.023} C_VEL
LIN {X 0,Y 592.036,Z 357.518,A -85,B 0,C 180,E1 28568.791,E2 28568.791} C_VEL
LIN {X 0,Y 593.825,Z 361.935,A -85,B 0,C 180,E1 28568.352,E2 28568.352} C_VEL
LIN {X 0,Y 595.141,Z 364.942,A -85,B 0,C 180,E1 28568.207,E2 28568.207} C_VEL
LIN {X 0,Y 594.77,Z 549.978,A -85,B 0,C 180,E1 28565.497,E2 28565.497} C_VEL
LIN {X 0,Y 594.41,Z 709.409,A -85,B 0,C 180,E1 28563.205,E2 28563.205} C_VEL
LIN {X 0,Y 594.249,Z 733.198,A -85,B 0,C 180,E1 28562.679,E2 28562.679} C_VEL
LIN {X 0,Y 594.111,Z 753.208,A -85,B 0,C 180,E1 28562.077,E2 28562.077} C_VEL
LIN {X 0,Y 593.86,Z 776.629,A -85,B 0,C 180,E1 28561.181,E2 28561.181} C_VEL
LIN {X 0,Y 593.679,Z 796.844,A -85,B 0,C 180,E1 28560.232,E2 28560.232} C_VEL
LIN {X 0,Y 593.396,Z 818.577,A -85,B 0,C 180,E1 28559.014,E2 28559.014} C_VEL
LIN {X 0,Y 593.18,Z 839.126,A -85,B 0,C 180,E1 28557.666,E2 28557.666} C_VEL
LIN {X 0,Y 592.925,Z 858.071,A -85,B 0,C 180,E1 28556.216,E2 28556.216} C_VEL
LIN {X 0,Y 592.677,Z 877.469,A -85,B 0,C 180,E1 28554.516,E2 28554.516} C_VEL
LIN {X 0,Y 592.526,Z 894.772,A -85,B 0,C 180,E1 28552.782,E2 28552.782} C_VEL
LIN {X 0,Y 592.351,Z 910.494,A -85,B 0,C 180,E1 28550.965,E2 28550.965} C_VEL
LIN {X 0,Y 592.195,Z 926.035,A -85,B 0,C 180,E1 28548.913,E2 28548.913} C_VEL
LIN {X 0,Y 592.108,Z 938.747,A -85,B 0,C 180,E1 28546.984,E2 28546.984} C_VEL
LIN {X 0,Y 592.028,Z 950.091,A -85,B 0,C 180,E1 28544.973,E2 28544.973} C_VEL
LIN {X 0,Y 591.975,Z 959.939,A -85,B 0,C 180,E1 28542.95,E2 28542.95} C_VEL
LIN {X 0,Y 591.923,Z 968.536,A -85,B 0,C 180,E1 28540.805,E2 28540.805} C_VEL
LIN {X 0,Y 591.925,Z 975.341,A -85,B 0,C 180,E1 28538.743,E2 28538.743} C_VEL
LIN {X 0,Y 591.913,Z 980.953,A -85,B 0,C 180,E1 28536.497,E2 28536.497} C_VEL
LIN {X 0,Y 591.906,Z 984.84,A -85,B 0,C 180,E1 28534.359,E2 28534.359} C_VEL
LIN {X 0,Y 591.915,Z 987.158,A -85,B 0,C 180,E1 28532.129,E2 28532.129} C_VEL
LIN {X 0,Y 591.911,Z 987.996,A -85,B 0,C 180,E1 28530,E2 28530} C_VEL
LIN {X 0,Y 591.915,Z 987.22,A -85,B 0,C 180,E1 28527.87,E2 28527.87} C_VEL
LIN {X 0,Y 591.904,Z 984.982,A -85,B 0,C 180,E1 28525.641,E2 28525.641} C_VEL
LIN {X 0,Y 591.92,Z 981.143,A -85,B 0,C 180,E1 28523.502,E2 28523.502} C_VEL
LIN {X 0,Y 591.92,Z 975.903,A -85,B 0,C 180,E1 28521.354,E2 28521.354} C_VEL
LIN {X 0,Y 591.919,Z 968.859,A -85,B 0,C 180,E1 28519.194,E2 28519.194} C_VEL
LIN {X 0,Y 591.98,Z 960.658,A -85,B 0,C 180,E1 28517.119,E2 28517.119} C_VEL
LIN {X 0,Y 592.023,Z 950.552,A -85,B 0,C 180,E1 28515.026,E2 28515.026} C_VEL
LIN {X 0,Y 592.101,Z 939.308,A -85,B 0,C 180,E1 28513.016,E2 28513.016} C_VEL
LIN {X 0,Y 592.192,Z 926.654,A -85,B 0,C 180,E1 28511.086,E2 28511.086} C_VEL
LIN {X 0,Y 592.345,Z 912.082,A -85,B 0,C 180,E1 28509.138,E2 28509.138} C_VEL
LIN {X 0,Y 592.487,Z 896.502,A -85,B 0,C 180,E1 28507.321,E2 28507.321} C_VEL
LIN {X 0,Y 592.671,Z 879.506,A -85,B 0,C 180,E1 28505.589,E2 28505.589} C_VEL
LIN {X 0,Y 592.91,Z 861.452,A -85,B 0,C 180,E1 28503.968,E2 28503.968} C_VEL
LIN {X 0,Y 593.101,Z 842.522,A -85,B 0,C 180,E1 28502.493,E2 28502.493} C_VEL
LIN {X 0,Y 593.377,Z 821.594,A -85,B 0,C 180,E1 28501.082,E2 28501.082} C_VEL
LIN {X 0,Y 593.602,Z 801.712,A -85,B 0,C 180,E1 28499.93,E2 28499.93} C_VEL
LIN {X 0,Y 593.844,Z 780.045,A -85,B 0,C 180,E1 28498.879,E2 28498.879} C_VEL
LIN {X 0,Y 594.02,Z 759.868,A -85,B 0,C 180,E1 28498.062,E2 28498.062} C_VEL
LIN {X 0,Y 594.231,Z 737.082,A -85,B 0,C 180,E1 28497.337,E2 28497.337} C_VEL
LIN {X 0,Y 594.352,Z 716.677,A -85,B 0,C 180,E1 28496.843,E2 28496.843} C_VEL
LIN {X 0,Y 594.483,Z 687.204,A -85,B 0,C 180,E1 28496.365,E2 28496.365} C_VEL
LIN {X 0,Y 594.933,Z 476.951,A -85,B 0,C 180,E1 28493.356,E2 28493.356} C_VEL
LIN {X 0,Y 595.025,Z 364.432,A -85,B 0,C 180,E1 28491.687,E2 28491.687} C_VEL
LIN {X 0,Y 593.483,Z 361.027,A -85,B 0,C 180,E1 28491.495,E2 28491.495} C_VEL
LIN {X 0,Y 592.055,Z 357.602,A -85,B 0,C 180,E1 28491.127,E2 28491.127} C_VEL
LIN {X 0,Y 592.018,Z 357.301,A -85,B 0,C 180,E1 28490.977,E2 28490.977} C_VEL
LIN {X 0,Y 592.026,Z 357.305,A -85,B 0,C 180,E1 28487.64,E2 28487.64} C_VEL
LIN {X 0,Y 592.034,Z 357.298,A -85,B 0,C 180,E1 28484.362,E2 28484.362} C_VEL
LIN {X 0,Y 592.003,Z 357.302,A -85,B 0,C 180,E1 28481.133,E2 28481.133} C_VEL
LIN {X 0,Y 592.032,Z 357.298,A -85,B 0,C 180,E1 28477.933,E2 28477.933} C_VEL
LIN {X 0,Y 591.994,Z 357.296,A -85,B 0,C 180,E1 28474.811,E2 28474.811} C_VEL
LIN {X 0,Y 592.035,Z 357.303,A -85,B 0,C 180,E1 28471.67,E2 28471.67} C_VEL
LIN {X 0,Y 591.99,Z 357.298,A -85,B 0,C 180,E1 28468.554,E2 28468.554} C_VEL
LIN {X 0,Y 592.031,Z 357.302,A -85,B 0,C 180,E1 28465.295,E2 28465.295} C_VEL
LIN {X 0,Y 591.991,Z 357.298,A -85,B 0,C 180,E1 28462.23,E2 28462.23} C_VEL
LIN {X 0,Y 592.002,Z 357.302,A -85,B 0,C 180,E1 28458.922,E2 28458.922} C_VEL
LIN {X 0,Y 591.997,Z 357.297,A -85,B 0,C 180,E1 28455.879,E2 28455.879} C_VEL
LIN {X 0,Y 591.981,Z 357.303,A -85,B 0,C 180,E1 28452.585,E2 28452.585} C_VEL
LIN {X 0,Y 591.999,Z 357.301,A -85,B 0,C 180,E1 28449.626,E2 28449.626} C_VEL
LIN {X 0,Y 591.974,Z 357.304,A -85,B 0,C 180,E1 28446.401,E2 28446.401} C_VEL
LIN {X 0,Y 591.989,Z 357.302,A -85,B 0,C 180,E1 28443.486,E2 28443.486} C_VEL
LIN {X 0,Y 591.968,Z 357.305,A -85,B 0,C 180,E1 28440.291,E2 28440.291} C_VEL
LIN {X 0,Y 591.968,Z 357.303,A -85,B 0,C 180,E1 28437.483,E2 28437.483} C_VEL
LIN {X 0,Y 591.96,Z 357.304,A -85,B 0,C 180,E1 28434.125,E2 28434.125} C_VEL
LIN {X 0,Y 591.958,Z 357.306,A -85,B 0,C 180,E1 28431.354,E2 28431.354} C_VEL
LIN {X 0,Y 591.963,Z 357.305,A -85,B 0,C 180,E1 28428.01,E2 28428.01} C_VEL
LIN {X 0,Y 591.964,Z 357.305,A -85,B 0,C 180,E1 28425.224,E2 28425.224} C_VEL
LIN {X 0,Y 591.975,Z 357.301,A -85,B 0,C 180,E1 28421.894,E2 28421.894} C_VEL
LIN {X 0,Y 591.971,Z 357.305,A -85,B 0,C 180,E1 28419.056,E2 28419.056} C_VEL
LIN {X 0,Y 591.985,Z 357.3,A -85,B 0,C 180,E1 28415.769,E2 28415.769} C_VEL
LIN {X 0,Y 591.98,Z 357.305,A -85,B 0,C 180,E1 28412.869,E2 28412.869} C_VEL
LIN {X 0,Y 591.99,Z 357.301,A -85,B 0,C 180,E1 28409.557,E2 28409.557} C_VEL
LIN {X 0,Y 592.001,Z 357.304,A -85,B 0,C 180,E1 28406.538,E2 28406.538} C_VEL
LIN {X 0,Y 591.988,Z 357.301,A -85,B 0,C 180,E1 28403.281,E2 28403.281} C_VEL
LIN {X 0,Y 592.027,Z 357.304,A -85,B 0,C 180,E1 28400.202,E2 28400.202} C_VEL
LIN {X 0,Y 591.989,Z 357.301,A -85,B 0,C 180,E1 28396.973,E2 28396.973} C_VEL
LIN {X 0,Y 592.038,Z 357.305,A -85,B 0,C 180,E1 28393.852,E2 28393.852} C_VEL
LIN {X 0,Y 592.014,Z 357.41,A -85,B 0,C 180,E1 28390.906,E2 28390.906} C_VEL
LIN {X 0,Y 593.388,Z 360.917,A -85,B 0,C 180,E1 28390.542,E2 28390.542} C_VEL
LIN {X 0,Y 594.653,Z 364.145,A -85,B 0,C 180,E1 28390.21,E2 28390.21} C_VEL
LIN {X 0,Y 594.537,Z 391.464,A -85,B 0,C 180,E1 28388.35,E2 28388.35} C_VEL
LIN {X 0,Y 595.21,Z 395.869,A -85,B 0,C 180,E1 28388.232,E2 28388.232} C_VEL
LIN {X 0,Y 594.723,Z 605.114,A -85,B 0,C 180,E1 28385.181,E2 28385.181} C_VEL
LIN {X 0,Y 594.412,Z 739.477,A -85,B 0,C 180,E1 28383.249,E2 28383.249} C_VEL
LIN {X 0,Y 594.249,Z 763.139,A -85,B 0,C 180,E1 28382.725,E2 28382.725} C_VEL
LIN {X 0,Y 594.112,Z 783.15,A -85,B 0,C 180,E1 28382.124,E2 28382.124} C_VEL
LIN {X 0,Y 593.86,Z 806.485,A -85,B 0,C 180,E1 28381.232,E2 28381.232} C_VEL
LIN {X 0,Y 593.681,Z 826.615,A -85,B 0,C 180,E1 28380.288,E2 28380.288} C_VEL
LIN {X 0,Y 593.398,Z 848.197,A -85,B 0,C 180,E1 28379.082,E2 28379.082} C_VEL
LIN {X 0,Y 593.193,Z 868.454,A -85,B 0,C 180,E1 28377.76,E2 28377.76} C_VEL
LIN {X 0,Y 592.925,Z 888.022,A -85,B 0,C 180,E1 28376.265,E2 28376.265} C_VEL
LIN {X 0,Y 592.682,Z 907.143,A -85,B 0,C 180,E1 28374.593,E2 28374.593} C_VEL
LIN {X 0,Y 592.532,Z 924.278,A -85,B 0,C 180,E1 28372.879,E2 28372.879} C_VEL
LIN {X 0,Y 592.349,Z 940.384,A -85,B 0,C 180,E1 28371.024,E2 28371.024} C_VEL
LIN {X 0,Y 592.194,Z 955.714,A -85,B 0,C 180,E1 28369.004,E2 28369.004} C_VEL
LIN {X 0,Y 592.107,Z 968.389,A -85,B 0,C 180,E1 28367.085,E2 28367.085} C_VEL
LIN {X 0,Y 592.025,Z 980.321,A -85,B 0,C 180,E1 28364.974,E2 28364.974} C_VEL
LIN {X 0,Y 591.979,Z 990.463,A -85,B 0,C 180,E1 28362.881,E2 28362.881} C_VEL
LIN {X 0,Y 591.921,Z 998.697,A -85,B 0,C 180,E1 28360.806,E2 28360.806} C_VEL
LIN {X 0,Y 591.922,Z 1005.777,A -85,B 0,C 180,E1 28358.646,E2 28358.646} C_VEL
LIN {X 0,Y 591.919,Z 1011.048,A -85,B 0,C 180,E1 28356.498,E2 28356.498} C_VEL
LIN {X 0,Y 591.905,Z 1014.913,A -85,B 0,C 180,E1 28354.359,E2 28354.359} C_VEL
LIN {X 0,Y 591.915,Z 1017.189,A -85,B 0,C 180,E1 28352.13,E2 28352.13} C_VEL
LIN {X 0,Y 591.909,Z 1018,A -85,B 0,C 180,E1 28350,E2 28350} C_VEL
LIN {X 0,Y 591.915,Z 1017.189,A -85,B 0,C 180,E1 28347.871,E2 28347.871} C_VEL
LIN {X 0,Y 591.905,Z 1014.914,A -85,B 0,C 180,E1 28345.641,E2 28345.641} C_VEL
LIN {X 0,Y 591.918,Z 1011.049,A -85,B 0,C 180,E1 28343.503,E2 28343.503} C_VEL
LIN {X 0,Y 591.923,Z 1005.48,A -85,B 0,C 180,E1 28341.257,E2 28341.257} C_VEL
LIN {X 0,Y 591.921,Z 998.698,A -85,B 0,C 180,E1 28339.195,E2 28339.195} C_VEL
LIN {X 0,Y 591.98,Z 990.465,A -85,B 0,C 180,E1 28337.12,E2 28337.12} C_VEL
LIN {X 0,Y 592.026,Z 980.304,A -85,B 0,C 180,E1 28335.023,E2 28335.023} C_VEL
LIN {X 0,Y 592.108,Z 968.26,A -85,B 0,C 180,E1 28332.894,E2 28332.894} C_VEL
LIN {X 0,Y 592.195,Z 955.638,A -85,B 0,C 180,E1 28330.985,E2 28330.985} C_VEL
LIN {X 0,Y 592.348,Z 940.384,A -85,B 0,C 180,E1 28328.976,E2 28328.976} C_VEL
LIN {X 0,Y 592.532,Z 924.28,A -85,B 0,C 180,E1 28327.122,E2 28327.122} C_VEL
LIN {X 0,Y 592.688,Z 906.832,A -85,B 0,C 180,E1 28325.378,E2 28325.378} C_VEL
LIN {X 0,Y 592.924,Z 888.028,A -85,B 0,C 180,E1 28323.735,E2 28323.735} C_VEL
LIN {X 0,Y 593.193,Z 868.453,A -85,B 0,C 180,E1 28322.24,E2 28322.24} C_VEL
LIN {X 0,Y 593.398,Z 848.207,A -85,B 0,C 180,E1 28320.919,E2 28320.919} C_VEL
LIN {X 0,Y 593.682,Z 826.628,A -85,B 0,C 180,E1 28319.712,E2 28319.712} C_VEL
LIN {X 0,Y 593.86,Z 806.499,A -85,B 0,C 180,E1 28318.768,E2 28318.768} C_VEL
LIN {X 0,Y 594.111,Z 783.17,A -85,B 0,C 180,E1 28317.877,E2 28317.877} C_VEL
LIN {X 0,Y 594.25,Z 763.138,A -85,B 0,C 180,E1 28317.275,E2 28317.275} C_VEL
LIN {X 0,Y 594.413,Z 739.176,A -85,B 0,C 180,E1 28316.746,E2 28316.746} C_VEL
LIN {X 0,Y 594.91,Z 515.138,A -85,B 0,C 180,E1 28313.52,E2 28313.52} C_VEL
LIN {X 0,Y 595.051,Z 393.771,A -85,B 0,C 180,E1 28311.724,E2 28311.724} C_VEL
LIN {X 0,Y 594.428,Z 390.608,A -85,B 0,C 180,E1 28311.613,E2 28311.613} C_VEL
LIN {X 0,Y 594.626,Z 363.811,A -85,B 0,C 180,E1 28309.764,E2 28309.764} C_VEL
LIN {X 0,Y 592.065,Z 357.742,A -85,B 0,C 180,E1 28309.122,E2 28309.122} C_VEL
LIN {X 0,Y 592.002,Z 357.304,A -85,B 0,C 180,E1 28309.063,E2 28309.063} C_VEL
LIN {X 0,Y 592.009,Z 357.3,A -85,B 0,C 180,E1 28305.733,E2 28305.733} C_VEL
LIN {X 0,Y 592.02,Z 357.299,A -85,B 0,C 180,E1 28302.586,E2 28302.586} C_VEL
LIN {X 0,Y 591.989,Z 357.304,A -85,B 0,C 180,E1 28299.334,E2 28299.334} C_VEL
LIN {X 0,Y 592.03,Z 357.3,A -85,B 0,C 180,E1 28296.235,E2 28296.235} C_VEL
LIN {X 0,Y 591.978,Z 357.302,A -85,B 0,C 180,E1 28293.062,E2 28293.062} C_VEL
LIN {X 0,Y 592.042,Z 357.299,A -85,B 0,C 180,E1 28289.973,E2 28289.973} C_VEL
LIN {X 0,Y 591.97,Z 357.303,A -85,B 0,C 180,E1 28286.806,E2 28286.806} C_VEL
LIN {X 0,Y 592.04,Z 357.299,A -85,B 0,C 180,E1 28283.699,E2 28283.699} C_VEL
LIN {X 0,Y 591.963,Z 357.304,A -85,B 0,C 180,E1 28280.568,E2 28280.568} C_VEL
LIN {X 0,Y 592.036,Z 357.299,A -85,B 0,C 180,E1 28277.43,E2 28277.43} C_VEL
LIN {X 0,Y 591.955,Z 357.305,A -85,B 0,C 180,E1 28274.376,E2 28274.376} C_VEL
LIN {X 0,Y 592.033,Z 357.306,A -85,B 0,C 180,E1 28271.297,E2 28271.297} C_VEL
LIN {X 0,Y 591.948,Z 357.305,A -85,B 0,C 180,E1 28268.234,E2 28268.234} C_VEL
LIN {X 0,Y 592.024,Z 357.306,A -85,B 0,C 180,E1 28265.135,E2 28265.135} C_VEL
LIN {X 0,Y 591.95,Z 357.304,A -85,B 0,C 180,E1 28262.129,E2 28262.129} C_VEL
LIN {X 0,Y 592.037,Z 357.304,A -85,B 0,C 180,E1 28259.032,E2 28259.032} C_VEL
LIN {X 0,Y 591.957,Z 357.304,A -85,B 0,C 180,E1 28255.932,E2 28255.932} C_VEL
LIN {X 0,Y 592.037,Z 357.303,A -85,B 0,C 180,E1 28252.821,E2 28252.821} C_VEL
LIN {X 0,Y 591.97,Z 357.303,A -85,B 0,C 180,E1 28250.018,E2 28250.018} C_VEL
LIN {X 0,Y 590.981,Z 357.431,A -85,B 0,C 180,E1 28249.272,E2 28249.272} C_VEL
LIN {X 0,Y 584.553,Z 358.241,A -85,B 0,C 180,E1 28247.126,E2 28247.126} C_VEL
LIN {X 0,Y 584.099,Z 358.291,A -85,B 0,C 180,E1 28246.635,E2 28246.635} C_VEL
LIN {X 0,Y 584.033,Z 358.289,A -85,B 0,C 180,E1 28243.592,E2 28243.592} C_VEL
LIN {X 0,Y 584.101,Z 358.291,A -85,B 0,C 180,E1 28240.5,E2 28240.5} C_VEL
LIN {X 0,Y 584.041,Z 358.29,A -85,B 0,C 180,E1 28237.344,E2 28237.344} C_VEL
LIN {X 0,Y 584.094,Z 358.288,A -85,B 0,C 180,E1 28234.118,E2 28234.118} C_VEL
LIN {X 0,Y 584.051,Z 358.29,A -85,B 0,C 180,E1 28231.009,E2 28231.009} C_VEL
LIN {X 0,Y 584.077,Z 358.288,A -85,B 0,C 180,E1 28227.717,E2 28227.717} C_VEL
LIN {X 0,Y 584.082,Z 358.287,A -85,B 0,C 180,E1 28224.527,E2 28224.527} C_VEL
LIN {X 0,Y 584.064,Z 358.285,A -85,B 0,C 180,E1 28221.309,E2 28221.309} C_VEL
LIN {X 0,Y 584.095,Z 358.292,A -85,B 0,C 180,E1 28218.117,E2 28218.117} C_VEL
LIN {X 0,Y 584.061,Z 358.291,A -85,B 0,C 180,E1 28214.868,E2 28214.868} C_VEL
LIN {X 0,Y 584.093,Z 358.292,A -85,B 0,C 180,E1 28211.725,E2 28211.725} C_VEL
LIN {X 0,Y 584.104,Z 358.346,A -85,B 0,C 180,E1 28209.356,E2 28209.356} C_VEL
LIN {X 0,Y 585.533,Z 361.989,A -85,B 0,C 180,E1 28208.997,E2 28208.997} C_VEL
LIN {X 0,Y 588.908,Z 367.878,A -85,B 0,C 180,E1 28208.641,E2 28208.641} C_VEL
LIN {X 0,Y 588.179,Z 575.46,A -85,B 0,C 180,E1 28205.581,E2 28205.581} C_VEL
LIN {X 0,Y 587.708,Z 709.56,A -85,B 0,C 180,E1 28203.632,E2 28203.632} C_VEL
LIN {X 0,Y 587.464,Z 733.357,A -85,B 0,C 180,E1 28203.101,E2 28203.101} C_VEL
LIN {X 0,Y 587.251,Z 753.878,A -85,B 0,C 180,E1 28202.476,E2 28202.476} C_VEL
LIN {X 0,Y 586.878,Z 776.818,A -85,B 0,C 180,E1 28201.587,E2 28201.587} C_VEL
LIN {X 0,Y 586.594,Z 797.662,A -85,B 0,C 180,E1 28200.596,E2 28200.596} C_VEL
LIN {X 0,Y 586.179,Z 818.386,A -85,B 0,C 180,E1 28199.419,E2 28199.419} C_VEL
LIN {X 0,Y 585.866,Z 838.691,A -85,B 0,C 180,E1 28198.075,E2 28198.075} C_VEL
LIN {X 0,Y 585.463,Z 858.081,A -85,B 0,C 180,E1 28196.576,E2 28196.576} C_VEL
LIN {X 0,Y 585.109,Z 877.505,A -85,B 0,C 180,E1 28194.852,E2 28194.852} C_VEL
LIN {X 0,Y 584.857,Z 894.666,A -85,B 0,C 180,E1 28193.11,E2 28193.11} C_VEL
LIN {X 0,Y 584.577,Z 910.765,A -85,B 0,C 180,E1 28191.225,E2 28191.225} C_VEL
LIN {X 0,Y 584.351,Z 926.041,A -85,B 0,C 180,E1 28189.177,E2 28189.177} C_VEL
LIN {X 0,Y 584.216,Z 938.749,A -85,B 0,C 180,E1 28187.22,E2 28187.22} C_VEL
LIN {X 0,Y 584.089,Z 950.616,A -85,B 0,C 180,E1 28185.08,E2 28185.08} C_VEL
LIN {X 0,Y 584.01,Z 960.703,A -85,B 0,C 180,E1 28182.959,E2 28182.959} C_VEL
LIN {X 0,Y 583.939,Z 968.895,A -85,B 0,C 180,E1 28180.855,E2 28180.855} C_VEL
LIN {X 0,Y 583.932,Z 975.927,A -85,B 0,C 180,E1 28178.665,E2 28178.665} C_VEL
LIN {X 0,Y 583.916,Z 981.162,A -85,B 0,C 180,E1 28176.488,E2 28176.488} C_VEL
LIN {X 0,Y 583.913,Z 985.112,A -85,B 0,C 180,E1 28174.222,E2 28174.222} C_VEL
LIN {X 0,Y 583.914,Z 987.226,A -85,B 0,C 180,E1 28172.06,E2 28172.06} C_VEL
LIN {X 0,Y 583.903,Z 987.972,A -85,B 0,C 180,E1 28169.804,E2 28169.804} C_VEL
LIN {X 0,Y 583.914,Z 987.153,A -85,B 0,C 180,E1 28167.743,E2 28167.743} C_VEL
LIN {X 0,Y 583.898,Z 984.827,A -85,B 0,C 180,E1 28165.482,E2 28165.482} C_VEL
LIN {X 0,Y 583.914,Z 981.142,A -85,B 0,C 180,E1 28163.413,E2 28163.413} C_VEL
LIN {X 0,Y 583.929,Z 975.901,A -85,B 0,C 180,E1 28161.235,E2 28161.235} C_VEL
LIN {X 0,Y 583.933,Z 968.858,A -85,B 0,C 180,E1 28159.045,E2 28159.045} C_VEL
LIN {X 0,Y 584.008,Z 960.656,A -85,B 0,C 180,E1 28156.94,E2 28156.94} C_VEL
LIN {X 0,Y 584.087,Z 950.553,A -85,B 0,C 180,E1 28154.818,E2 28154.818} C_VEL
LIN {X 0,Y 584.212,Z 938.667,A -85,B 0,C 180,E1 28152.677,E2 28152.677} C_VEL
LIN {X 0,Y 584.348,Z 925.943,A -85,B 0,C 180,E1 28150.719,E2 28150.719} C_VEL
LIN {X 0,Y 584.576,Z 910.373,A -85,B 0,C 180,E1 28148.637,E2 28148.637} C_VEL
LIN {X 0,Y 584.858,Z 894.591,A -85,B 0,C 180,E1 28146.792,E2 28146.792} C_VEL
LIN {X 0,Y 585.116,Z 877.287,A -85,B 0,C 180,E1 28145.037,E2 28145.037} C_VEL
LIN {X 0,Y 585.465,Z 857.84,A -85,B 0,C 180,E1 28143.314,E2 28143.314} C_VEL
LIN {X 0,Y 585.861,Z 838.85,A -85,B 0,C 180,E1 28141.846,E2 28141.846} C_VEL
LIN {X 0,Y 586.173,Z 818.914,A -85,B 0,C 180,E1 28140.524,E2 28140.524} C_VEL
LIN {X 0,Y 586.597,Z 797.503,A -85,B 0,C 180,E1 28139.307,E2 28139.307} C_VEL
LIN {X 0,Y 586.871,Z 777.487,A -85,B 0,C 180,E1 28138.353,E2 28138.353} C_VEL
LIN {X 0,Y 587.245,Z 754.709,A -85,B 0,C 180,E1 28137.462,E2 28137.462} C_VEL
LIN {X 0,Y 587.459,Z 733.855,A -85,B 0,C 180,E1 28136.823,E2 28136.823} C_VEL
LIN {X 0,Y 587.706,Z 710.653,A -85,B 0,C 180,E1 28136.296,E2 28136.296} C_VEL
LIN {X 0,Y 587.956,Z 642.252,A -85,B 0,C 180,E1 28135.291,E2 28135.291} C_VEL
LIN {X 0,Y 588.648,Z 435.529,A -85,B 0,C 180,E1 28132.277,E2 28132.277} C_VEL
LIN {X 0,Y 588.798,Z 367.377,A -85,B 0,C 180,E1 28131.252,E2 28131.252} C_VEL
LIN {X 0,Y 584.928,Z 360.983,A -85,B 0,C 180,E1 28130.823,E2 28130.823} C_VEL
LIN {X 0,Y 584.094,Z 358.291,A -85,B 0,C 180,E1 28130.536,E2 28130.536} C_VEL
LIN {X 0,Y 584.07,Z 358.293,A -85,B 0,C 180,E1 28127.326,E2 28127.326} C_VEL
LIN {X 0,Y 584.09,Z 358.29,A -85,B 0,C 180,E1 28124.164,E2 28124.164} C_VEL
LIN {X 0,Y 584.064,Z 358.29,A -85,B 0,C 180,E1 28120.97,E2 28120.97} C_VEL
LIN {X 0,Y 584.096,Z 358.289,A -85,B 0,C 180,E1 28117.743,E2 28117.743} C_VEL
LIN {X 0,Y 584.061,Z 358.282,A -85,B 0,C 180,E1 28114.58,E2 28114.58} C_VEL
LIN {X 0,Y 584.075,Z 358.291,A -85,B 0,C 180,E1 28111.245,E2 28111.245} C_VEL
LIN {X 0,Y 584.083,Z 358.283,A -85,B 0,C 180,E1 28108.084,E2 28108.084} C_VEL
LIN {X 0,Y 584.05,Z 358.288,A -85,B 0,C 180,E1 28104.798,E2 28104.798} C_VEL
LIN {X 0,Y 584.098,Z 358.285,A -85,B 0,C 180,E1 28101.658,E2 28101.658} C_VEL
LIN {X 0,Y 584.04,Z 358.288,A -85,B 0,C 180,E1 28098.465,E2 28098.465} C_VEL
LIN {X 0,Y 584.1,Z 358.288,A -85,B 0,C 180,E1 28095.285,E2 28095.285} C_VEL
LIN {X 0,Y 584.034,Z 358.29,A -85,B 0,C 180,E1 28092.156,E2 28092.156} C_VEL
LIN {X 0,Y 584.087,Z 358.293,A -85,B 0,C 180,E1 28088.962,E2 28088.962} C_VEL
LIN {X 0,Y 584.03,Z 358.292,A -85,B 0,C 180,E1 28085.896,E2 28085.896} C_VEL
LIN {X 0,Y 584.06,Z 358.294,A -85,B 0,C 180,E1 28082.649,E2 28082.649} C_VEL
LIN {X 0,Y 584.023,Z 358.293,A -85,B 0,C 180,E1 28079.706,E2 28079.706} C_VEL
LIN {X 0,Y 584.05,Z 358.295,A -85,B 0,C 180,E1 28076.467,E2 28076.467} C_VEL
LIN {X 0,Y 584.012,Z 358.293,A -85,B 0,C 180,E1 28073.611,E2 28073.611} C_VEL
LIN {X 0,Y 584.061,Z 358.294,A -85,B 0,C 180,E1 28070.442,E2 28070.442} C_VEL
LIN {X 0,Y 584.012,Z 358.294,A -85,B 0,C 180,E1 28067.543,E2 28067.543} C_VEL
LIN {X 0,Y 584.087,Z 358.291,A -85,B 0,C 180,E1 28064.41,E2 28064.41} C_VEL
LIN {X 0,Y 584.021,Z 358.289,A -85,B 0,C 180,E1 28061.328,E2 28061.328} C_VEL
LIN {X 0,Y 584.088,Z 358.289,A -85,B 0,C 180,E1 28058.194,E2 28058.194} C_VEL
LIN {X 0,Y 584.028,Z 358.29,A -85,B 0,C 180,E1 28055.13,E2 28055.13} C_VEL
LIN {X 0,Y 584.078,Z 358.286,A -85,B 0,C 180,E1 28051.917,E2 28051.917} C_VEL
LIN {X 0,Y 584.041,Z 358.292,A -85,B 0,C 180,E1 28048.868,E2 28048.868} C_VEL
LIN {X 0,Y 584.068,Z 358.287,A -85,B 0,C 180,E1 28045.592,E2 28045.592} C_VEL
LIN {X 0,Y 584.055,Z 358.293,A -85,B 0,C 180,E1 28042.575,E2 28042.575} C_VEL
LIN {X 0,Y 584.063,Z 358.289,A -85,B 0,C 180,E1 28039.29,E2 28039.29} C_VEL
LIN {X 0,Y 584.09,Z 358.295,A -85,B 0,C 180,E1 28036.104,E2 28036.104} C_VEL
LIN {X 0,Y 584.054,Z 358.293,A -85,B 0,C 180,E1 28032.887,E2 28032.887} C_VEL
LIN {X 0,Y 584.102,Z 358.315,A -85,B 0,C 180,E1 28031.516,E2 28031.516} C_VEL
LIN {X 0,Y 585.466,Z 361.897,A -85,B 0,C 180,E1 28031.137,E2 28031.137} C_VEL
LIN {X 0,Y 588.044,Z 367.725,A -85,B 0,C 180,E1 28030.5,E2 28030.5} C_VEL
LIN {X 0,Y 587.863,Z 391.498,A -85,B 0,C 180,E1 28028.866,E2 28028.866} C_VEL
LIN {X 0,Y 588.914,Z 397.411,A -85,B 0,C 180,E1 28028.693,E2 28028.693} C_VEL
LIN {X 0,Y 588.172,Z 607.202,A -85,B 0,C 180,E1 28025.601,E2 28025.601} C_VEL
LIN {X 0,Y 587.711,Z 739.585,A -85,B 0,C 180,E1 28023.676,E2 28023.676} C_VEL
LIN {X 0,Y 587.464,Z 763.316,A -85,B 0,C 180,E1 28023.147,E2 28023.147} C_VEL
LIN {X 0,Y 587.251,Z 783.907,A -85,B 0,C 180,E1 28022.52,E2 28022.52} C_VEL
LIN {X 0,Y 586.873,Z 807.171,A -85,B 0,C 180,E1 28021.616,E2 28021.616} C_VEL
LIN {X 0,Y 586.588,Z 828.56,A -85,B 0,C 180,E1 28020.595,E2 28020.595} C_VEL
LIN {X 0,Y 586.171,Z 849.091,A -85,B 0,C 180,E1 28019.42,E2 28019.42} C_VEL
LIN {X 0,Y 585.845,Z 869.344,A -85,B 0,C 180,E1 28018.072,E2 28018.072} C_VEL
LIN {X 0,Y 585.465,Z 887.958,A -85,B 0,C 180,E1 28016.632,E2 28016.632} C_VEL
LIN {X 0,Y 585.121,Z 907.124,A -85,B 0,C 180,E1 28014.934,E2 28014.934} C_VEL
LIN {X 0,Y 584.863,Z 924.146,A -85,B 0,C 180,E1 28013.21,E2 28013.21} C_VEL
LIN {X 0,Y 584.579,Z 940.009,A -85,B 0,C 180,E1 28011.363,E2 28011.363} C_VEL
LIN {X 0,Y 584.373,Z 954.927,A -85,B 0,C 180,E1 28009.384,E2 28009.384} C_VEL
LIN {X 0,Y 584.224,Z 967.748,A -85,B 0,C 180,E1 28007.426,E2 28007.426} C_VEL
LIN {X 0,Y 584.09,Z 979.802,A -85,B 0,C 180,E1 28005.283,E2 28005.283} C_VEL
LIN {X 0,Y 584.001,Z 989.546,A -85,B 0,C 180,E1 28003.262,E2 28003.262} C_VEL
LIN {X 0,Y 583.938,Z 998.341,A -85,B 0,C 180,E1 28001.055,E2 28001.055} C_VEL
LIN {X 0,Y 583.939,Z 1004.871,A -85,B 0,C 180,E1 27999.063,E2 27999.063} C_VEL
LIN {X 0,Y 583.898,Z 1010.635,A -85,B 0,C 180,E1 27996.785,E2 27996.785} C_VEL
LIN {X 0,Y 583.9,Z 1014.276,A -85,B 0,C 180,E1 27994.813,E2 27994.813} C_VEL
LIN {X 0,Y 583.916,Z 1016.987,A -85,B 0,C 180,E1 27992.453,E2 27992.453} C_VEL
LIN {X 0,Y 583.888,Z 1017.917,A -85,B 0,C 180,E1 27990.393,E2 27990.393} C_VEL
LIN {X 0,Y 583.912,Z 1017.324,A -85,B 0,C 180,E1 27988.038,E2 27988.038} C_VEL
LIN {X 0,Y 583.915,Z 1015.278,A -85,B 0,C 180,E1 27985.877,E2 27985.877} C_VEL
LIN {X 0,Y 583.923,Z 1011.462,A -85,B 0,C 180,E1 27983.611,E2 27983.611} C_VEL
LIN {X 0,Y 583.927,Z 1006.553,A -85,B 0,C 180,E1 27981.533,E2 27981.533} C_VEL
LIN {X 0,Y 583.939,Z 999.411,A -85,B 0,C 180,E1 27979.245,E2 27979.245} C_VEL
LIN {X 0,Y 584.007,Z 991.704,A -85,B 0,C 180,E1 27977.242,E2 27977.242} C_VEL
LIN {X 0,Y 584.082,Z 981.368,A -85,B 0,C 180,E1 27975.022,E2 27975.022} C_VEL
LIN {X 0,Y 584.197,Z 970.247,A -85,B 0,C 180,E1 27972.985,E2 27972.985} C_VEL
LIN {X 0,Y 584.339,Z 957.057,A -85,B 0,C 180,E1 27970.927,E2 27970.927} C_VEL
LIN {X 0,Y 584.566,Z 942.565,A -85,B 0,C 180,E1 27968.952,E2 27968.952} C_VEL
LIN {X 0,Y 584.787,Z 927.42,A -85,B 0,C 180,E1 27967.156,E2 27967.156} C_VEL
LIN {X 0,Y 585.065,Z 909.673,A -85,B 0,C 180,E1 27965.312,E2 27965.312} C_VEL
LIN {X 0,Y 585.425,Z 892.251,A -85,B 0,C 180,E1 27963.721,E2 27963.721} C_VEL
LIN {X 0,Y 585.727,Z 873.384,A -85,B 0,C 180,E1 27962.227,E2 27962.227} C_VEL
LIN {X 0,Y 586.143,Z 851.77,A -85,B 0,C 180,E1 27960.748,E2 27960.748} C_VEL
LIN {X 0,Y 586.501,Z 831.913,A -85,B 0,C 180,E1 27959.585,E2 27959.585} C_VEL
LIN {X 0,Y 586.849,Z 810.319,A -85,B 0,C 180,E1 27958.524,E2 27958.524} C_VEL
LIN {X 0,Y 587.149,Z 789.634,A -85,B 0,C 180,E1 27957.68,E2 27957.68} C_VEL
LIN {X 0,Y 587.441,Z 766.904,A -85,B 0,C 180,E1 27956.952,E2 27956.952} C_VEL
LIN {X 0,Y 587.629,Z 745.843,A -85,B 0,C 180,E1 27956.44,E2 27956.44} C_VEL
LIN {X 0,Y 587.82,Z 714.803,A -85,B 0,C 180,E1 27955.943,E2 27955.943} C_VEL
LIN {X 0,Y 588.501,Z 507.123,A -85,B 0,C 180,E1 27952.937,E2 27952.937} C_VEL
LIN {X 0,Y 588.74,Z 395.533,A -85,B 0,C 180,E1 27951.265,E2 27951.265} C_VEL
LIN {X 0,Y 587.746,Z 390.733,A -85,B 0,C 180,E1 27951.103,E2 27951.103} C_VEL
LIN {X 0,Y 587.961,Z 367.495,A -85,B 0,C 180,E1 27949.477,E2 27949.477} C_VEL
LIN {X 0,Y 584.144,Z 358.596,A -85,B 0,C 180,E1 27948.508,E2 27948.508} C_VEL
LIN {X 0,Y 584.098,Z 358.293,A -85,B 0,C 180,E1 27948.387,E2 27948.387} C_VEL
LIN {X 0,Y 584.051,Z 358.288,A -85,B 0,C 180,E1 27945.271,E2 27945.271} C_VEL
LIN {X 0,Y 584.099,Z 358.287,A -85,B 0,C 180,E1 27942.146,E2 27942.146} C_VEL
LIN {X 0,Y 584.046,Z 358.291,A -85,B 0,C 180,E1 27939.001,E2 27939.001} C_VEL
LIN {X 0,Y 584.094,Z 358.293,A -85,B 0,C 180,E1 27935.777,E2 27935.777} C_VEL
LIN {X 0,Y 584.04,Z 358.29,A -85,B 0,C 180,E1 27932.75,E2 27932.75} C_VEL
LIN {X 0,Y 584.081,Z 358.287,A -85,B 0,C 180,E1 27929.538,E2 27929.538} C_VEL
LIN {X 0,Y 584.035,Z 358.291,A -85,B 0,C 180,E1 27926.54,E2 27926.54} C_VEL
LIN {X 0,Y 584.065,Z 358.291,A -85,B 0,C 180,E1 27923.294,E2 27923.294} C_VEL
LIN {X 0,Y 584.031,Z 358.292,A -85,B 0,C 180,E1 27920.336,E2 27920.336} C_VEL
LIN {X 0,Y 584.045,Z 358.29,A -85,B 0,C 180,E1 27917.022,E2 27917.022} C_VEL
LIN {X 0,Y 584.023,Z 358.294,A -85,B 0,C 180,E1 27914.171,E2 27914.171} C_VEL
LIN {X 0,Y 584.049,Z 358.295,A -85,B 0,C 180,E1 27910.954,E2 27910.954} C_VEL
LIN {X 0,Y 584.012,Z 358.294,A -85,B 0,C 180,E1 27908.07,E2 27908.07} C_VEL
LIN {X 0,Y 584.059,Z 358.295,A -85,B 0,C 180,E1 27904.91,E2 27904.91} C_VEL
LIN {X 0,Y 584.014,Z 358.293,A -85,B 0,C 180,E1 27901.962,E2 27901.962} C_VEL
LIN {X 0,Y 584.078,Z 358.291,A -85,B 0,C 180,E1 27898.823,E2 27898.823} C_VEL
LIN {X 0,Y 584.022,Z 358.294,A -85,B 0,C 180,E1 27895.778,E2 27895.778} C_VEL
LIN {X 0,Y 584.08,Z 358.291,A -85,B 0,C 180,E1 27892.623,E2 27892.623} C_VEL
LIN {X 0,Y 584.028,Z 358.293,A -85,B 0,C 180,E1 27889.644,E2 27889.644} C_VEL
LIN {X 0,Y 584.099,Z 358.291,A -85,B 0,C 180,E1 27886.635,E2 27886.635} C_VEL
LIN {X 0,Y 583.064,Z 358.416,A -85,B 0,C 180,E1 27885.88,E2 27885.88} C_VEL
LIN {X 0,Y 576.61,Z 359.214,A -85,B 0,C 180,E1 27883.76,E2 27883.76} C_VEL
LIN {X 0,Y 576.108,Z 359.278,A -85,B 0,C 180,E1 27883.207,E2 27883.207} C_VEL
LIN {X 0,Y 576.111,Z 359.279,A -85,B 0,C 180,E1 27879.853,E2 27879.853} C_VEL
LIN {X 0,Y 576.137,Z 359.278,A -85,B 0,C 180,E1 27876.799,E2 27876.799} C_VEL
LIN {X 0,Y 576.109,Z 359.279,A -85,B 0,C 180,E1 27873.51,E2 27873.51} C_VEL
LIN {X 0,Y 576.161,Z 359.273,A -85,B 0,C 180,E1 27870.358,E2 27870.358} C_VEL
LIN {X 0,Y 576.112,Z 359.28,A -85,B 0,C 180,E1 27867.097,E2 27867.097} C_VEL
LIN {X 0,Y 576.159,Z 359.276,A -85,B 0,C 180,E1 27863.841,E2 27863.841} C_VEL
LIN {X 0,Y 576.133,Z 359.276,A -85,B 0,C 180,E1 27860.567,E2 27860.567} C_VEL
LIN {X 0,Y 576.131,Z 359.278,A -85,B 0,C 180,E1 27857.224,E2 27857.224} C_VEL
LIN {X 0,Y 576.157,Z 359.274,A -85,B 0,C 180,E1 27854.073,E2 27854.073} C_VEL
LIN {X 0,Y 576.127,Z 359.281,A -85,B 0,C 180,E1 27850.828,E2 27850.828} C_VEL
LIN {X 0,Y 576.188,Z 359.503,A -85,B 0,C 180,E1 27849.914,E2 27849.914} C_VEL
LIN {X 0,Y 577.111,Z 362.202,A -85,B 0,C 180,E1 27849.675,E2 27849.675} C_VEL
LIN {X 0,Y 582.643,Z 371.135,A -85,B 0,C 180,E1 27849.086,E2 27849.086} C_VEL
LIN {X 0,Y 581.655,Z 579.165,A -85,B 0,C 180,E1 27845.988,E2 27845.988} C_VEL
LIN {X 0,Y 581.039,Z 709.817,A -85,B 0,C 180,E1 27844.067,E2 27844.067} C_VEL
LIN {X 0,Y 580.71,Z 733.644,A -85,B 0,C 180,E1 27843.529,E2 27843.529} C_VEL
LIN {X 0,Y 580.416,Z 754.872,A -85,B 0,C 180,E1 27842.873,E2 27842.873} C_VEL
LIN {X 0,Y 579.924,Z 777.583,A -85,B 0,C 180,E1 27841.976,E2 27841.976} C_VEL
LIN {X 0,Y 579.523,Z 799.103,A -85,B 0,C 180,E1 27840.936,E2 27840.936} C_VEL
LIN {X 0,Y 578.958,Z 820.4,A -85,B 0,C 180,E1 27839.694,E2 27839.694} C_VEL
LIN {X 0,Y 578.475,Z 841.341,A -85,B 0,C 180,E1 27838.264,E2 27838.264} C_VEL
LIN {X 0,Y 577.997,Z 859.885,A -85,B 0,C 180,E1 27836.796,E2 27836.796} C_VEL
LIN {X 0,Y 577.532,Z 878.59,A -85,B 0,C 180,E1 27835.094,E2 27835.094} C_VEL
LIN {X 0,Y 577.177,Z 895.46,A -85,B 0,C 180,E1 27833.345,E2 27833.345} C_VEL
LIN {X 0,Y 576.811,Z 911.359,A -85,B 0,C 180,E1 27831.451,E2 27831.451} C_VEL
LIN {X 0,Y 576.512,Z 926.658,A -85,B 0,C 180,E1 27829.357,E2 27829.357} C_VEL
LIN {X 0,Y 576.323,Z 939.386,A -85,B 0,C 180,E1 27827.359,E2 27827.359} C_VEL
LIN {X 0,Y 576.151,Z 950.948,A -85,B 0,C 180,E1 27825.228,E2 27825.228} C_VEL
LIN {X 0,Y 576.039,Z 961.116,A -85,B 0,C 180,E1 27823.039,E2 27823.039} C_VEL
LIN {X 0,Y 575.956,Z 968.898,A -85,B 0,C 180,E1 27821.007,E2 27821.007} C_VEL
LIN {X 0,Y 575.946,Z 975.647,A -85,B 0,C 180,E1 27818.887,E2 27818.887} C_VEL
LIN {X 0,Y 575.904,Z 980.956,A -85,B 0,C 180,E1 27816.679,E2 27816.679} C_VEL
LIN {X 0,Y 575.903,Z 984.842,A -85,B 0,C 180,E1 27814.48,E2 27814.48} C_VEL
LIN {X 0,Y 575.915,Z 987.159,A -85,B 0,C 180,E1 27812.188,E2 27812.188} C_VEL
LIN {X 0,Y 575.911,Z 987.996,A -85,B 0,C 180,E1 27810,E2 27810} C_VEL
LIN {X 0,Y 575.915,Z 987.219,A -85,B 0,C 180,E1 27807.811,E2 27807.811} C_VEL
LIN {X 0,Y 575.901,Z 984.98,A -85,B 0,C 180,E1 27805.519,E2 27805.519} C_VEL
LIN {X 0,Y 575.909,Z 981.141,A -85,B 0,C 180,E1 27803.321,E2 27803.321} C_VEL
LIN {X 0,Y 575.94,Z 975.9,A -85,B 0,C 180,E1 27801.112,E2 27801.112} C_VEL
LIN {X 0,Y 575.95,Z 969.213,A -85,B 0,C 180,E1 27798.992,E2 27798.992} C_VEL
LIN {X 0,Y 576.037,Z 961.474,A -85,B 0,C 180,E1 27796.96,E2 27796.96} C_VEL
LIN {X 0,Y 576.146,Z 951.412,A -85,B 0,C 180,E1 27794.774,E2 27794.774} C_VEL
LIN {X 0,Y 576.31,Z 939.914,A -85,B 0,C 180,E1 27792.64,E2 27792.64} C_VEL
LIN {X 0,Y 576.494,Z 927.302,A -85,B 0,C 180,E1 27790.648,E2 27790.648} C_VEL
LIN {X 0,Y 576.792,Z 912.915,A -85,B 0,C 180,E1 27788.654,E2 27788.654} C_VEL
LIN {X 0,Y 577.115,Z 897.574,A -85,B 0,C 180,E1 27786.808,E2 27786.808} C_VEL
LIN {X 0,Y 577.487,Z 880.046,A -85,B 0,C 180,E1 27784.958,E2 27784.958} C_VEL
LIN {X 0,Y 577.971,Z 861.805,A -85,B 0,C 180,E1 27783.273,E2 27783.273} C_VEL
LIN {X 0,Y 578.436,Z 842.508,A -85,B 0,C 180,E1 27781.733,E2 27781.733} C_VEL
LIN {X 0,Y 578.941,Z 821.577,A -85,B 0,C 180,E1 27780.29,E2 27780.29} C_VEL
LIN {X 0,Y 579.442,Z 801.677,A -85,B 0,C 180,E1 27779.116,E2 27779.116} C_VEL
LIN {X 0,Y 579.892,Z 779.705,A -85,B 0,C 180,E1 27778.029,E2 27778.029} C_VEL
LIN {X 0,Y 580.342,Z 758.603,A -85,B 0,C 180,E1 27777.168,E2 27777.168} C_VEL
LIN {X 0,Y 580.688,Z 736.009,A -85,B 0,C 180,E1 27776.447,E2 27776.447} C_VEL
LIN {X 0,Y 581,Z 713.849,A -85,B 0,C 180,E1 27775.915,E2 27775.915} C_VEL
LIN {X 0,Y 581.229,Z 675.989,A -85,B 0,C 180,E1 27775.328,E2 27775.328} C_VEL
LIN {X 0,Y 582.191,Z 463.61,A -85,B 0,C 180,E1 27772.215,E2 27772.215} C_VEL
LIN {X 0,Y 582.526,Z 370.782,A -85,B 0,C 180,E1 27770.81,E2 27770.81} C_VEL
LIN {X 0,Y 576.687,Z 361.33,A -85,B 0,C 180,E1 27770.181,E2 27770.181} C_VEL
LIN {X 0,Y 576.155,Z 359.283,A -85,B 0,C 180,E1 27769.962,E2 27769.962} C_VEL
LIN {X 0,Y 576.156,Z 359.277,A -85,B 0,C 180,E1 27766.596,E2 27766.596} C_VEL
LIN {X 0,Y 576.131,Z 359.281,A -85,B 0,C 180,E1 27763.276,E2 27763.276} C_VEL
LIN {X 0,Y 576.155,Z 359.278,A -85,B 0,C 180,E1 27760.073,E2 27760.073} C_VEL
LIN {X 0,Y 576.121,Z 359.279,A -85,B 0,C 180,E1 27756.872,E2 27756.872} C_VEL
LIN {X 0,Y 576.158,Z 359.274,A -85,B 0,C 180,E1 27753.603,E2 27753.603} C_VEL
LIN {X 0,Y 576.125,Z 359.275,A -85,B 0,C 180,E1 27750.408,E2 27750.408} C_VEL
LIN {X 0,Y 576.125,Z 359.282,A -85,B 0,C 180,E1 27747.046,E2 27747.046} C_VEL
LIN {X 0,Y 576.152,Z 359.271,A -85,B 0,C 180,E1 27743.851,E2 27743.851} C_VEL
LIN {X 0,Y 576.106,Z 359.281,A -85,B 0,C 180,E1 27740.629,E2 27740.629} C_VEL
LIN {X 0,Y 576.16,Z 359.273,A -85,B 0,C 180,E1 27737.471,E2 27737.471} C_VEL
LIN {X 0,Y 576.097,Z 359.281,A -85,B 0,C 180,E1 27734.37,E2 27734.37} C_VEL
LIN {X 0,Y 576.162,Z 359.279,A -85,B 0,C 180,E1 27731.208,E2 27731.208} C_VEL
LIN {X 0,Y 576.091,Z 359.279,A -85,B 0,C 180,E1 27728.082,E2 27728.082} C_VEL
LIN {X 0,Y 576.145,Z 359.282,A -85,B 0,C 180,E1 27724.878,E2 27724.878} C_VEL
LIN {X 0,Y 576.085,Z 359.281,A -85,B 0,C 180,E1 27721.79,E2 27721.79} C_VEL
LIN {X 0,Y 576.124,Z 359.282,A -85,B 0,C 180,E1 27718.608,E2 27718.608} C_VEL
LIN {X 0,Y 576.078,Z 359.283,A -85,B 0,C 180,E1 27715.62,E2 27715.62} C_VEL
LIN {X 0,Y 576.114,Z 359.284,A -85,B 0,C 180,E1 27712.421,E2 27712.421} C_VEL
LIN {X 0,Y 576.076,Z 359.283,A -85,B 0,C 180,E1 27709.399,E2 27709.399} C_VEL
LIN {X 0,Y 576.105,Z 359.283,A -85,B 0,C 180,E1 27706.143,E2 27706.143} C_VEL
LIN {X 0,Y 576.083,Z 359.28,A -85,B 0,C 180,E1 27703.255,E2 27703.255} C_VEL
LIN {X 0,Y 576.116,Z 359.282,A -85,B 0,C 180,E1 27700.008,E2 27700.008} C_VEL
LIN {X 0,Y 576.096,Z 359.28,A -85,B 0,C 180,E1 27697.014,E2 27697.014} C_VEL
LIN {X 0,Y 576.104,Z 359.281,A -85,B 0,C 180,E1 27693.622,E2 27693.622} C_VEL
LIN {X 0,Y 576.113,Z 359.277,A -85,B 0,C 180,E1 27690.698,E2 27690.698} C_VEL
LIN {X 0,Y 576.111,Z 359.278,A -85,B 0,C 180,E1 27687.452,E2 27687.452} C_VEL
LIN {X 0,Y 576.142,Z 359.281,A -85,B 0,C 180,E1 27684.331,E2 27684.331} C_VEL
LIN {X 0,Y 576.107,Z 359.277,A -85,B 0,C 180,E1 27681.078,E2 27681.078} C_VEL
LIN {X 0,Y 576.161,Z 359.274,A -85,B 0,C 180,E1 27677.944,E2 27677.944} C_VEL
LIN {X 0,Y 576.112,Z 359.281,A -85,B 0,C 180,E1 27674.779,E2 27674.779} C_VEL
LIN {X 0,Y 576.142,Z 359.293,A -85,B 0,C 180,E1 27672.147,E2 27672.147} C_VEL
LIN {X 0,Y 577.585,Z 362.941,A -85,B 0,C 180,E1 27671.746,E2 27671.746} C_VEL
LIN {X 0,Y 581.431,Z 371.306,A -85,B 0,C 180,E1 27670.798,E2 27670.798} C_VEL
LIN {X 0,Y 581.219,Z 391.52,A -85,B 0,C 180,E1 27669.395,E2 27669.395} C_VEL
LIN {X 0,Y 582.657,Z 399.179,A -85,B 0,C 180,E1 27669.16,E2 27669.16} C_VEL
LIN {X 0,Y 581.651,Z 609.873,A -85,B 0,C 180,E1 27666.023,E2 27666.023} C_VEL
LIN {X 0,Y 581.04,Z 739.799,A -85,B 0,C 180,E1 27664.112,E2 27664.112} C_VEL
LIN {X 0,Y 580.711,Z 763.616,A -85,B 0,C 180,E1 27663.574,E2 27663.574} C_VEL
LIN {X 0,Y 580.417,Z 784.825,A -85,B 0,C 180,E1 27662.92,E2 27662.92} C_VEL
LIN {X 0,Y 579.949,Z 806.492,A -85,B 0,C 180,E1 27662.07,E2 27662.07} C_VEL
LIN {X 0,Y 579.542,Z 827.739,A -85,B 0,C 180,E1 27661.051,E2 27661.051} C_VEL
LIN {X 0,Y 578.992,Z 849.094,A -85,B 0,C 180,E1 27659.821,E2 27659.821} C_VEL
LIN {X 0,Y 578.528,Z 869.793,A -85,B 0,C 180,E1 27658.425,E2 27658.425} C_VEL
LIN {X 0,Y 578.018,Z 888.621,A -85,B 0,C 180,E1 27656.947,E2 27656.947} C_VEL
LIN {X 0,Y 577.554,Z 907.932,A -85,B 0,C 180,E1 27655.203,E2 27655.203} C_VEL
LIN {X 0,Y 577.192,Z 924.959,A -85,B 0,C 180,E1 27653.448,E2 27653.448} C_VEL
LIN {X 0,Y 576.815,Z 940.862,A -85,B 0,C 180,E1 27651.558,E2 27651.558} C_VEL
LIN {X 0,Y 576.518,Z 956.346,A -85,B 0,C 180,E1 27649.448,E2 27649.448} C_VEL
LIN {X 0,Y 576.323,Z 969.344,A -85,B 0,C 180,E1 27647.411,E2 27647.411} C_VEL
LIN {X 0,Y 576.149,Z 980.845,A -85,B 0,C 180,E1 27645.293,E2 27645.293} C_VEL
LIN {X 0,Y 576.036,Z 990.885,A -85,B 0,C 180,E1 27643.142,E2 27643.142} C_VEL
LIN {X 0,Y 575.955,Z 998.698,A -85,B 0,C 180,E1 27641.109,E2 27641.109} C_VEL
LIN {X 0,Y 575.945,Z 1005.559,A -85,B 0,C 180,E1 27638.961,E2 27638.961} C_VEL
LIN {X 0,Y 575.908,Z 1011.048,A -85,B 0,C 180,E1 27636.679,E2 27636.679} C_VEL
LIN {X 0,Y 575.901,Z 1014.913,A -85,B 0,C 180,E1 27634.481,E2 27634.481} C_VEL
LIN {X 0,Y 575.915,Z 1017.189,A -85,B 0,C 180,E1 27632.189,E2 27632.189} C_VEL
LIN {X 0,Y 575.909,Z 1018,A -85,B 0,C 180,E1 27630,E2 27630} C_VEL
LIN {X 0,Y 575.915,Z 1017.189,A -85,B 0,C 180,E1 27627.812,E2 27627.812} C_VEL
LIN {X 0,Y 575.901,Z 1014.914,A -85,B 0,C 180,E1 27625.52,E2 27625.52} C_VEL
LIN {X 0,Y 575.907,Z 1011.049,A -85,B 0,C 180,E1 27623.321,E2 27623.321} C_VEL
LIN {X 0,Y 575.944,Z 1005.56,A -85,B 0,C 180,E1 27621.039,E2 27621.039} C_VEL
LIN {X 0,Y 575.955,Z 998.7,A -85,B 0,C 180,E1 27618.891,E2 27618.891} C_VEL
LIN {X 0,Y 576.039,Z 990.464,A -85,B 0,C 180,E1 27616.757,E2 27616.757} C_VEL
LIN {X 0,Y 576.149,Z 980.849,A -85,B 0,C 180,E1 27614.707,E2 27614.707} C_VEL
LIN {X 0,Y 576.323,Z 969.346,A -85,B 0,C 180,E1 27612.589,E2 27612.589} C_VEL
LIN {X 0,Y 576.518,Z 956.35,A -85,B 0,C 180,E1 27610.552,E2 27610.552} C_VEL
LIN {X 0,Y 576.814,Z 940.867,A -85,B 0,C 180,E1 27608.442,E2 27608.442} C_VEL
LIN {X 0,Y 577.198,Z 924.703,A -85,B 0,C 180,E1 27606.524,E2 27606.524} C_VEL
LIN {X 0,Y 577.573,Z 907.386,A -85,B 0,C 180,E1 27604.744,E2 27604.744} C_VEL
LIN {X 0,Y 578.038,Z 887.681,A -85,B 0,C 180,E1 27602.975,E2 27602.975} C_VEL
LIN {X 0,Y 578.574,Z 868.241,A -85,B 0,C 180,E1 27601.46,E2 27601.46} C_VEL
LIN {X 0,Y 579.038,Z 847.693,A -85,B 0,C 180,E1 27600.092,E2 27600.092} C_VEL
LIN {X 0,Y 579.565,Z 825.51,A -85,B 0,C 180,E1 27598.836,E2 27598.836} C_VEL
LIN {X 0,Y 579.992,Z 805.225,A -85,B 0,C 180,E1 27597.875,E2 27597.875} C_VEL
LIN {X 0,Y 580.438,Z 782.315,A -85,B 0,C 180,E1 27596.996,E2 27596.996} C_VEL
LIN {X 0,Y 580.745,Z 761.454,A -85,B 0,C 180,E1 27596.366,E2 27596.366} C_VEL
LIN {X 0,Y 581.049,Z 738.188,A -85,B 0,C 180,E1 27595.86,E2 27595.86} C_VEL
LIN {X 0,Y 582.058,Z 518.7,A -85,B 0,C 180,E1 27592.632,E2 27592.632} C_VEL
LIN {X 0,Y 582.506,Z 397.421,A -85,B 0,C 180,E1 27590.801,E2 27590.801} C_VEL
LIN {X 0,Y 581.097,Z 390.56,A -85,B 0,C 180,E1 27590.56,E2 27590.56} C_VEL
LIN {X 0,Y 581.347,Z 371.084,A -85,B 0,C 180,E1 27589.178,E2 27589.178} C_VEL
LIN {X 0,Y 576.191,Z 359.622,A -85,B 0,C 180,E1 27587.882,E2 27587.882} C_VEL
LIN {X 0,Y 576.135,Z 359.285,A -85,B 0,C 180,E1 27587.814,E2 27587.814} C_VEL
LIN {X 0,Y 576.143,Z 359.273,A -85,B 0,C 180,E1 27584.648,E2 27584.648} C_VEL
LIN {X 0,Y 576.114,Z 359.282,A -85,B 0,C 180,E1 27581.394,E2 27581.394} C_VEL
LIN {X 0,Y 576.163,Z 359.279,A -85,B 0,C 180,E1 27578.155,E2 27578.155} C_VEL
LIN {X 0,Y 576.101,Z 359.277,A -85,B 0,C 180,E1 27574.941,E2 27574.941} C_VEL
LIN {X 0,Y 576.156,Z 359.283,A -85,B 0,C 180,E1 27571.723,E2 27571.723} C_VEL
LIN {X 0,Y 576.094,Z 359.275,A -85,B 0,C 180,E1 27568.734,E2 27568.734} C_VEL
LIN {X 0,Y 576.15,Z 359.279,A -85,B 0,C 180,E1 27565.537,E2 27565.537} C_VEL
LIN {X 0,Y 576.09,Z 359.277,A -85,B 0,C 180,E1 27562.447,E2 27562.447} C_VEL
LIN {X 0,Y 576.129,Z 359.278,A -85,B 0,C 180,E1 27559.253,E2 27559.253} C_VEL
LIN {X 0,Y 576.082,Z 359.278,A -85,B 0,C 180,E1 27556.325,E2 27556.325} C_VEL
LIN {X 0,Y 576.128,Z 359.282,A -85,B 0,C 180,E1 27553.141,E2 27553.141} C_VEL
LIN {X 0,Y 576.074,Z 359.283,A -85,B 0,C 180,E1 27550.197,E2 27550.197} C_VEL
LIN {X 0,Y 576.122,Z 359.283,A -85,B 0,C 180,E1 27546.978,E2 27546.978} C_VEL
LIN {X 0,Y 576.073,Z 359.284,A -85,B 0,C 180,E1 27543.981,E2 27543.981} C_VEL
LIN {X 0,Y 576.124,Z 359.283,A -85,B 0,C 180,E1 27540.795,E2 27540.795} C_VEL
LIN {X 0,Y 576.081,Z 359.281,A -85,B 0,C 180,E1 27537.811,E2 27537.811} C_VEL
LIN {X 0,Y 576.131,Z 359.28,A -85,B 0,C 180,E1 27534.622,E2 27534.622} C_VEL
LIN {X 0,Y 576.09,Z 359.282,A -85,B 0,C 180,E1 27531.617,E2 27531.617} C_VEL
LIN {X 0,Y 576.13,Z 359.278,A -85,B 0,C 180,E1 27528.386,E2 27528.386} C_VEL
LIN {X 0,Y 576.103,Z 359.282,A -85,B 0,C 180,E1 27525.322,E2 27525.322} C_VEL
LIN {X 0,Y 576.108,Z 359.278,A -85,B 0,C 180,E1 27523.207,E2 27523.207} C_VEL
LIN {X 0,Y 575.161,Z 359.402,A -85,B 0,C 180,E1 27522.441,E2 27522.441} C_VEL
LIN {X 0,Y 568.621,Z 360.216,A -85,B 0,C 180,E1 27520.235,E2 27520.235} C_VEL
LIN {X 0,Y 568.166,Z 360.269,A -85,B 0,C 180,E1 27519.731,E2 27519.731} C_VEL
LIN {X 0,Y 568.219,Z 360.259,A -85,B 0,C 180,E1 27516.567,E2 27516.567} C_VEL
LIN {X 0,Y 568.167,Z 360.269,A -85,B 0,C 180,E1 27513.336,E2 27513.336} C_VEL
LIN {X 0,Y 568.222,Z 360.26,A -85,B 0,C 180,E1 27510.134,E2 27510.134} C_VEL
LIN {X 0,Y 568.181,Z 360.271,A -85,B 0,C 180,E1 27506.881,E2 27506.881} C_VEL
LIN {X 0,Y 568.194,Z 360.266,A -85,B 0,C 180,E1 27503.503,E2 27503.503} C_VEL
LIN {X 0,Y 568.218,Z 360.262,A -85,B 0,C 180,E1 27500.252,E2 27500.252} C_VEL
LIN {X 0,Y 568.183,Z 360.269,A -85,B 0,C 180,E1 27496.939,E2 27496.939} C_VEL
LIN {X 0,Y 568.216,Z 360.255,A -85,B 0,C 180,E1 27493.679,E2 27493.679} C_VEL
LIN {X 0,Y 568.207,Z 360.396,A -85,B 0,C 180,E1 27490.52,E2 27490.52} C_VEL
LIN {X 0,Y 568.773,Z 362.413,A -85,B 0,C 180,E1 27490.373,E2 27490.373} C_VEL
LIN {X 0,Y 575.856,Z 373.319,A -85,B 0,C 180,E1 27489.603,E2 27489.603} C_VEL
LIN {X 0,Y 576.409,Z 374.935,A -85,B 0,C 180,E1 27489.531,E2 27489.531} C_VEL
LIN {X 0,Y 575.155,Z 583.658,A -85,B 0,C 180,E1 27486.392,E2 27486.392} C_VEL
LIN {X 0,Y 574.404,Z 709.968,A -85,B 0,C 180,E1 27484.514,E2 27484.514} C_VEL
LIN {X 0,Y 573.996,Z 733.722,A -85,B 0,C 180,E1 27483.973,E2 27483.973} C_VEL
LIN {X 0,Y 573.617,Z 755.327,A -85,B 0,C 180,E1 27483.298,E2 27483.298} C_VEL
LIN {X 0,Y 573.053,Z 776.815,A -85,B 0,C 180,E1 27482.443,E2 27482.443} C_VEL
LIN {X 0,Y 572.514,Z 798.016,A -85,B 0,C 180,E1 27481.416,E2 27481.416} C_VEL
LIN {X 0,Y 571.849,Z 819.305,A -85,B 0,C 180,E1 27480.174,E2 27480.174} C_VEL
LIN {X 0,Y 571.24,Z 839.879,A -85,B 0,C 180,E1 27478.769,E2 27478.769} C_VEL
LIN {X 0,Y 570.612,Z 858.763,A -85,B 0,C 180,E1 27477.268,E2 27477.268} C_VEL
LIN {X 0,Y 570.05,Z 877.492,A -85,B 0,C 180,E1 27475.558,E2 27475.558} C_VEL
LIN {X 0,Y 569.549,Z 894.791,A -85,B 0,C 180,E1 27473.756,E2 27473.756} C_VEL
LIN {X 0,Y 569.093,Z 910.515,A -85,B 0,C 180,E1 27471.865,E2 27471.865} C_VEL
LIN {X 0,Y 568.717,Z 926.054,A -85,B 0,C 180,E1 27469.725,E2 27469.725} C_VEL
LIN {X 0,Y 568.447,Z 938.754,A -85,B 0,C 180,E1 27467.713,E2 27467.713} C_VEL
LIN {X 0,Y 568.216,Z 950.626,A -85,B 0,C 180,E1 27465.511,E2 27465.511} C_VEL
LIN {X 0,Y 568.075,Z 960.709,A -85,B 0,C 180,E1 27463.329,E2 27463.329} C_VEL
LIN {X 0,Y 567.978,Z 968.901,A -85,B 0,C 180,E1 27461.164,E2 27461.164} C_VEL
LIN {X 0,Y 567.956,Z 975.649,A -85,B 0,C 180,E1 27459.013,E2 27459.013} C_VEL
LIN {X 0,Y 567.901,Z 980.958,A -85,B 0,C 180,E1 27456.773,E2 27456.773} C_VEL
LIN {X 0,Y 567.902,Z 984.684,A -85,B 0,C 180,E1 27454.645,E2 27454.645} C_VEL
LIN {X 0,Y 567.915,Z 987.092,A -85,B 0,C 180,E1 27452.32,E2 27452.32} C_VEL
LIN {X 0,Y 567.908,Z 987.974,A -85,B 0,C 180,E1 27450.101,E2 27450.101} C_VEL
LIN {X 0,Y 567.914,Z 987.219,A -85,B 0,C 180,E1 27447.78,E2 27447.78} C_VEL
LIN {X 0,Y 567.899,Z 984.979,A -85,B 0,C 180,E1 27445.456,E2 27445.456} C_VEL
LIN {X 0,Y 567.903,Z 981.108,A -85,B 0,C 180,E1 27443.211,E2 27443.211} C_VEL
LIN {X 0,Y 567.953,Z 975.867,A -85,B 0,C 180,E1 27440.975,E2 27440.975} C_VEL
LIN {X 0,Y 567.975,Z 968.855,A -85,B 0,C 180,E1 27438.733,E2 27438.733} C_VEL
LIN {X 0,Y 568.075,Z 960.651,A -85,B 0,C 180,E1 27436.567,E2 27436.567} C_VEL
LIN {X 0,Y 568.218,Z 950.549,A -85,B 0,C 180,E1 27434.383,E2 27434.383} C_VEL
LIN {X 0,Y 568.449,Z 938.655,A -85,B 0,C 180,E1 27432.18,E2 27432.18} C_VEL
LIN {X 0,Y 568.724,Z 925.806,A -85,B 0,C 180,E1 27430.147,E2 27430.147} C_VEL
LIN {X 0,Y 569.097,Z 910.365,A -85,B 0,C 180,E1 27428.026,E2 27428.026} C_VEL
LIN {X 0,Y 569.55,Z 894.782,A -85,B 0,C 180,E1 27426.153,E2 27426.153} C_VEL
LIN {X 0,Y 570.055,Z 877.273,A -85,B 0,C 180,E1 27424.33,E2 27424.33} C_VEL
LIN {X 0,Y 570.646,Z 857.827,A -85,B 0,C 180,E1 27422.563,E2 27422.563} C_VEL
LIN {X 0,Y 571.276,Z 838.792,A -85,B 0,C 180,E1 27421.058,E2 27421.058} C_VEL
LIN {X 0,Y 571.864,Z 818.899,A -85,B 0,C 180,E1 27419.711,E2 27419.711} C_VEL
LIN {X 0,Y 572.521,Z 797.303,A -85,B 0,C 180,E1 27418.457,E2 27418.457} C_VEL
LIN {X 0,Y 573.059,Z 776.653,A -85,B 0,C 180,E1 27417.46,E2 27417.46} C_VEL
LIN {X 0,Y 573.634,Z 753.486,A -85,B 0,C 180,E1 27416.549,E2 27416.549} C_VEL
LIN {X 0,Y 574.018,Z 732.462,A -85,B 0,C 180,E1 27415.903,E2 27415.903} C_VEL
LIN {X 0,Y 574.414,Z 708.834,A -85,B 0,C 180,E1 27415.377,E2 27415.377} C_VEL
LIN {X 0,Y 575.684,Z 491.181,A -85,B 0,C 180,E1 27412.14,E2 27412.14} C_VEL
LIN {X 0,Y 576.245,Z 374.024,A -85,B 0,C 180,E1 27410.351,E2 27410.351} C_VEL
LIN {X 0,Y 570.271,Z 364.711,A -85,B 0,C 180,E1 27409.702,E2 27409.702} C_VEL
LIN {X 0,Y 568.473,Z 361.574,A -85,B 0,C 180,E1 27409.497,E2 27409.497} C_VEL
LIN {X 0,Y 568.195,Z 360.273,A -85,B 0,C 180,E1 27409.348,E2 27409.348} C_VEL
LIN {X 0,Y 568.214,Z 360.27,A -85,B 0,C 180,E1 27406.114,E2 27406.114} C_VEL
LIN {X 0,Y 568.19,Z 360.268,A -85,B 0,C 180,E1 27402.923,E2 27402.923} C_VEL
LIN {X 0,Y 568.213,Z 360.262,A -85,B 0,C 180,E1 27399.568,E2 27399.568} C_VEL
LIN {X 0,Y 568.213,Z 360.265,A -85,B 0,C 180,E1 27396.245,E2 27396.245} C_VEL
LIN {X 0,Y 568.181,Z 360.269,A -85,B 0,C 180,E1 27392.933,E2 27392.933} C_VEL
LIN {X 0,Y 568.221,Z 360.262,A -85,B 0,C 180,E1 27389.75,E2 27389.75} C_VEL
LIN {X 0,Y 568.174,Z 360.269,A -85,B 0,C 180,E1 27386.55,E2 27386.55} C_VEL
LIN {X 0,Y 568.216,Z 360.26,A -85,B 0,C 180,E1 27383.302,E2 27383.302} C_VEL
LIN {X 0,Y 568.173,Z 360.268,A -85,B 0,C 180,E1 27380.177,E2 27380.177} C_VEL
LIN {X 0,Y 568.174,Z 360.264,A -85,B 0,C 180,E1 27376.775,E2 27376.775} C_VEL
LIN {X 0,Y 568.186,Z 360.268,A -85,B 0,C 180,E1 27373.743,E2 27373.743} C_VEL
LIN {X 0,Y 568.159,Z 360.271,A -85,B 0,C 180,E1 27370.443,E2 27370.443} C_VEL
LIN {X 0,Y 568.202,Z 360.266,A -85,B 0,C 180,E1 27367.381,E2 27367.381} C_VEL
LIN {X 0,Y 568.147,Z 360.27,A -85,B 0,C 180,E1 27364.138,E2 27364.138} C_VEL
LIN {X 0,Y 568.218,Z 360.268,A -85,B 0,C 180,E1 27361.008,E2 27361.008} C_VEL
LIN {X 0,Y 568.139,Z 360.27,A -85,B 0,C 180,E1 27357.882,E2 27357.882} C_VEL
LIN {X 0,Y 568.21,Z 360.27,A -85,B 0,C 180,E1 27354.75,E2 27354.75} C_VEL
LIN {X 0,Y 568.131,Z 360.273,A -85,B 0,C 180,E1 27351.703,E2 27351.703} C_VEL
LIN {X 0,Y 568.204,Z 360.271,A -85,B 0,C 180,E1 27348.531,E2 27348.531} C_VEL
LIN {X 0,Y 568.138,Z 360.273,A -85,B 0,C 180,E1 27345.424,E2 27345.424} C_VEL
LIN {X 0,Y 568.2,Z 360.261,A -85,B 0,C 180,E1 27342.277,E2 27342.277} C_VEL
LIN {X 0,Y 568.148,Z 360.273,A -85,B 0,C 180,E1 27339.177,E2 27339.177} C_VEL
LIN {X 0,Y 568.181,Z 360.265,A -85,B 0,C 180,E1 27335.905,E2 27335.905} C_VEL
LIN {X 0,Y 568.163,Z 360.272,A -85,B 0,C 180,E1 27332.885,E2 27332.885} C_VEL
LIN {X 0,Y 568.173,Z 360.268,A -85,B 0,C 180,E1 27329.548,E2 27329.548} C_VEL
LIN {X 0,Y 568.191,Z 360.267,A -85,B 0,C 180,E1 27326.458,E2 27326.458} C_VEL
LIN {X 0,Y 568.168,Z 360.269,A -85,B 0,C 180,E1 27323.189,E2 27323.189} C_VEL
LIN {X 0,Y 568.218,Z 360.272,A -85,B 0,C 180,E1 27320.039,E2 27320.039} C_VEL
LIN {X 0,Y 568.171,Z 360.27,A -85,B 0,C 180,E1 27316.758,E2 27316.758} C_VEL
LIN {X 0,Y 568.22,Z 360.269,A -85,B 0,C 180,E1 27313.467,E2 27313.467} C_VEL
LIN {X 0,Y 568.189,Z 360.378,A -85,B 0,C 180,E1 27312.794,E2 27312.794} C_VEL
LIN {X 0,Y 569.254,Z 363.396,A -85,B 0,C 180,E1 27312.464,E2 27312.464} C_VEL
LIN {X 0,Y 572.204,Z 369.516,A -85,B 0,C 180,E1 27311.735,E2 27311.735} C_VEL
LIN {X 0,Y 574.856,Z 375.406,A -85,B 0,C 180,E1 27311.063,E2 27311.063} C_VEL
LIN {X 0,Y 574.596,Z 391.45,A -85,B 0,C 180,E1 27309.941,E2 27309.941} C_VEL
LIN {X 0,Y 576.439,Z 400.866,A -85,B 0,C 180,E1 27309.638,E2 27309.638} C_VEL
LIN {X 0,Y 575.166,Z 611.935,A -85,B 0,C 180,E1 27306.462,E2 27306.462} C_VEL
LIN {X 0,Y 574.406,Z 739.907,A -85,B 0,C 180,E1 27304.56,E2 27304.56} C_VEL
LIN {X 0,Y 573.992,Z 763.771,A -85,B 0,C 180,E1 27304.016,E2 27304.016} C_VEL
LIN {X 0,Y 573.613,Z 785.657,A -85,B 0,C 180,E1 27303.332,E2 27303.332} C_VEL
LIN {X 0,Y 573.016,Z 807.768,A -85,B 0,C 180,E1 27302.446,E2 27302.446} C_VEL
LIN {X 0,Y 572.502,Z 828.856,A -85,B 0,C 180,E1 27301.417,E2 27301.417} C_VEL
LIN {X 0,Y 571.823,Z 849.987,A -85,B 0,C 180,E1 27300.176,E2 27300.176} C_VEL
LIN {X 0,Y 571.197,Z 871.113,A -85,B 0,C 180,E1 27298.721,E2 27298.721} C_VEL
LIN {X 0,Y 570.594,Z 889.285,A -85,B 0,C 180,E1 27297.27,E2 27297.27} C_VEL
LIN {X 0,Y 570.011,Z 908.486,A -85,B 0,C 180,E1 27295.505,E2 27295.505} C_VEL
LIN {X 0,Y 569.524,Z 925.639,A -85,B 0,C 180,E1 27293.703,E2 27293.703} C_VEL
LIN {X 0,Y 569.059,Z 941.711,A -85,B 0,C 180,E1 27291.759,E2 27291.759} C_VEL
LIN {X 0,Y 568.707,Z 956.348,A -85,B 0,C 180,E1 27289.726,E2 27289.726} C_VEL
LIN {X 0,Y 568.445,Z 969.019,A -85,B 0,C 180,E1 27287.714,E2 27287.714} C_VEL
LIN {X 0,Y 568.22,Z 980.325,A -85,B 0,C 180,E1 27285.617,E2 27285.617} C_VEL
LIN {X 0,Y 568.08,Z 990.003,A -85,B 0,C 180,E1 27283.537,E2 27283.537} C_VEL
LIN {X 0,Y 567.985,Z 998.483,A -85,B 0,C 180,E1 27281.329,E2 27281.329} C_VEL
LIN {X 0,Y 567.948,Z 1005.175,A -85,B 0,C 180,E1 27279.218,E2 27279.218} C_VEL
LIN {X 0,Y 567.895,Z 1010.635,A -85,B 0,C 180,E1 27276.977,E2 27276.977} C_VEL
LIN {X 0,Y 567.907,Z 1014.277,A -85,B 0,C 180,E1 27274.949,E2 27274.949} C_VEL
LIN {X 0,Y 567.914,Z 1016.988,A -85,B 0,C 180,E1 27272.523,E2 27272.523} C_VEL
LIN {X 0,Y 567.887,Z 1017.917,A -85,B 0,C 180,E1 27270.404,E2 27270.404} C_VEL
LIN {X 0,Y 567.913,Z 1017.324,A -85,B 0,C 180,E1 27267.983,E2 27267.983} C_VEL
LIN {X 0,Y 567.911,Z 1015.277,A -85,B 0,C 180,E1 27265.76,E2 27265.76} C_VEL
LIN {X 0,Y 567.92,Z 1011.463,A -85,B 0,C 180,E1 27263.43,E2 27263.43} C_VEL
LIN {X 0,Y 567.94,Z 1006.554,A -85,B 0,C 180,E1 27261.293,E2 27261.293} C_VEL
LIN {X 0,Y 567.969,Z 999.769,A -85,B 0,C 180,E1 27259.042,E2 27259.042} C_VEL
LIN {X 0,Y 568.067,Z 992.115,A -85,B 0,C 180,E1 27256.982,E2 27256.982} C_VEL
LIN {X 0,Y 568.211,Z 981.612,A -85,B 0,C 180,E1 27254.641,E2 27254.641} C_VEL
LIN {X 0,Y 568.423,Z 970.251,A -85,B 0,C 180,E1 27252.497,E2 27252.497} C_VEL
LIN {X 0,Y 568.669,Z 957.594,A -85,B 0,C 180,E1 27250.46,E2 27250.46} C_VEL
LIN {X 0,Y 569.029,Z 943.406,A -85,B 0,C 180,E1 27248.457,E2 27248.457} C_VEL
LIN {X 0,Y 569.447,Z 927.935,A -85,B 0,C 180,E1 27246.565,E2 27246.565} C_VEL
LIN {X 0,Y 569.949,Z 910.151,A -85,B 0,C 180,E1 27244.66,E2 27244.66} C_VEL
LIN {X 0,Y 570.535,Z 891.937,A -85,B 0,C 180,E1 27242.953,E2 27242.953} C_VEL
LIN {X 0,Y 571.138,Z 872.661,A -85,B 0,C 180,E1 27241.397,E2 27241.397} C_VEL
LIN {X 0,Y 571.757,Z 852.036,A -85,B 0,C 180,E1 27239.954,E2 27239.954} C_VEL
LIN {X 0,Y 572.398,Z 831.906,A -85,B 0,C 180,E1 27238.753,E2 27238.753} C_VEL
LIN {X 0,Y 572.972,Z 809.419,A -85,B 0,C 180,E1 27237.628,E2 27237.628} C_VEL
LIN {X 0,Y 573.578,Z 787.483,A -85,B 0,C 180,E1 27236.732,E2 27236.732} C_VEL
LIN {X 0,Y 573.978,Z 765.042,A -85,B 0,C 180,E1 27236.019,E2 27236.019} C_VEL
LIN {X 0,Y 574.392,Z 742.193,A -85,B 0,C 180,E1 27235.48,E2 27235.48} C_VEL
LIN {X 0,Y 574.737,Z 689.152,A -85,B 0,C 180,E1 27234.673,E2 27234.673} C_VEL
LIN {X 0,Y 575.98,Z 474.263,A -85,B 0,C 180,E1 27231.479,E2 27231.479} C_VEL
LIN {X 0,Y 576.257,Z 399.025,A -85,B 0,C 180,E1 27230.317,E2 27230.317} C_VEL
LIN {X 0,Y 574.492,Z 390.627,A -85,B 0,C 180,E1 27230.021,E2 27230.021} C_VEL
LIN {X 0,Y 574.766,Z 375.136,A -85,B 0,C 180,E1 27228.909,E2 27228.909} C_VEL
LIN {X 0,Y 569.729,Z 364.095,A -85,B 0,C 180,E1 27227.632,E2 27227.632} C_VEL
LIN {X 0,Y 568.219,Z 360.575,A -85,B 0,C 180,E1 27227.224,E2 27227.224} C_VEL
LIN {X 0,Y 568.18,Z 360.273,A -85,B 0,C 180,E1 27227.059,E2 27227.059} C_VEL
LIN {X 0,Y 568.193,Z 360.272,A -85,B 0,C 180,E1 27223.684,E2 27223.684} C_VEL
LIN {X 0,Y 568.205,Z 360.267,A -85,B 0,C 180,E1 27220.49,E2 27220.49} C_VEL
LIN {X 0,Y 568.169,Z 360.272,A -85,B 0,C 180,E1 27217.255,E2 27217.255} C_VEL
LIN {X 0,Y 568.222,Z 360.26,A -85,B 0,C 180,E1 27214.025,E2 27214.025} C_VEL
LIN {X 0,Y 568.16,Z 360.268,A -85,B 0,C 180,E1 27210.804,E2 27210.804} C_VEL
LIN {X 0,Y 568.21,Z 360.268,A -85,B 0,C 180,E1 27207.567,E2 27207.567} C_VEL
LIN {X 0,Y 568.152,Z 360.264,A -85,B 0,C 180,E1 27204.532,E2 27204.532} C_VEL
LIN {X 0,Y 568.199,Z 360.272,A -85,B 0,C 180,E1 27201.362,E2 27201.362} C_VEL
LIN {X 0,Y 568.151,Z 360.264,A -85,B 0,C 180,E1 27198.255,E2 27198.255} C_VEL
LIN {X 0,Y 568.158,Z 360.273,A -85,B 0,C 180,E1 27194.888,E2 27194.888} C_VEL
LIN {X 0,Y 568.153,Z 360.269,A -85,B 0,C 180,E1 27191.943,E2 27191.943} C_VEL
LIN {X 0,Y 568.142,Z 360.272,A -85,B 0,C 180,E1 27188.603,E2 27188.603} C_VEL
LIN {X 0,Y 568.157,Z 360.272,A -85,B 0,C 180,E1 27185.655,E2 27185.655} C_VEL
LIN {X 0,Y 568.143,Z 360.27,A -85,B 0,C 180,E1 27182.42,E2 27182.42} C_VEL
LIN {X 0,Y 568.164,Z 360.273,A -85,B 0,C 180,E1 27179.496,E2 27179.496} C_VEL
LIN {X 0,Y 568.147,Z 360.271,A -85,B 0,C 180,E1 27176.165,E2 27176.165} C_VEL
LIN {X 0,Y 568.194,Z 360.272,A -85,B 0,C 180,E1 27173.127,E2 27173.127} C_VEL
LIN {X 0,Y 568.153,Z 360.27,A -85,B 0,C 180,E1 27169.966,E2 27169.966} C_VEL
LIN {X 0,Y 568.211,Z 360.269,A -85,B 0,C 180,E1 27166.88,E2 27166.88} C_VEL
LIN {X 0,Y 568.156,Z 360.265,A -85,B 0,C 180,E1 27163.646,E2 27163.646} C_VEL
LIN {X 0,Y 568.223,Z 360.269,A -85,B 0,C 180,E1 27160.468,E2 27160.468} C_VEL
LIN {X 0,Y 568.166,Z 360.269,A -85,B 0,C 180,E1 27159.731,E2 27159.731} C_VEL
LIN {X 0,Y 567.181,Z 360.399,A -85,B 0,C 180,E1 27158.954,E2 27158.954} C_VEL
LIN {X 0,Y 560.747,Z 361.19,A -85,B 0,C 180,E1 27156.717,E2 27156.717} C_VEL
LIN {X 0,Y 560.277,Z 361.245,A -85,B 0,C 180,E1 27156.205,E2 27156.205} C_VEL
LIN {X 0,Y 560.236,Z 361.26,A -85,B 0,C 180,E1 27153.043,E2 27153.043} C_VEL
LIN {X 0,Y 560.25,Z 361.25,A -85,B 0,C 180,E1 27149.665,E2 27149.665} C_VEL
LIN {X 0,Y 560.276,Z 361.252,A -85,B 0,C 180,E1 27146.412,E2 27146.412} C_VEL
LIN {X 0,Y 560.239,Z 361.258,A -85,B 0,C 180,E1 27143.077,E2 27143.077} C_VEL
LIN {X 0,Y 560.284,Z 361.255,A -85,B 0,C 180,E1 27139.758,E2 27139.758} C_VEL
LIN {X 0,Y 560.263,Z 361.262,A -85,B 0,C 180,E1 27136.425,E2 27136.425} C_VEL
LIN {X 0,Y 560.255,Z 361.241,A -85,B 0,C 180,E1 27133.113,E2 27133.113} C_VEL
LIN {X 0,Y 560.292,Z 361.458,A -85,B 0,C 180,E1 27131.132,E2 27131.132} C_VEL
LIN {X 0,Y 561.575,Z 364.765,A -85,B 0,C 180,E1 27130.963,E2 27130.963} C_VEL
LIN {X 0,Y 563.631,Z 367.399,A -85,B 0,C 180,E1 27130.738,E2 27130.738} C_VEL
LIN {X 0,Y 570.217,Z 377.758,A -85,B 0,C 180,E1 27130.002,E2 27130.002} C_VEL
LIN {X 0,Y 568.694,Z 586.931,A -85,B 0,C 180,E1 27126.823,E2 27126.823} C_VEL
LIN {X 0,Y 567.805,Z 710.119,A -85,B 0,C 180,E1 27124.971,E2 27124.971} C_VEL
LIN {X 0,Y 567.319,Z 733.817,A -85,B 0,C 180,E1 27124.426,E2 27124.426} C_VEL
LIN {X 0,Y 566.851,Z 755.783,A -85,B 0,C 180,E1 27123.734,E2 27123.734} C_VEL
LIN {X 0,Y 566.148,Z 778.107,A -85,B 0,C 180,E1 27122.828,E2 27122.828} C_VEL
LIN {X 0,Y 565.497,Z 799.129,A -85,B 0,C 180,E1 27121.792,E2 27121.792} C_VEL
LIN {X 0,Y 564.748,Z 819.231,A -85,B 0,C 180,E1 27120.599,E2 27120.599} C_VEL
LIN {X 0,Y 563.979,Z 839.885,A -85,B 0,C 180,E1 27119.175,E2 27119.175} C_VEL
LIN {X 0,Y 563.267,Z 858.112,A -85,B 0,C 180,E1 27117.711,E2 27117.711} C_VEL
LIN {X 0,Y 562.544,Z 877.499,A -85,B 0,C 180,E1 27115.924,E2 27115.924} C_VEL
LIN {X 0,Y 561.916,Z 894.77,A -85,B 0,C 180,E1 27114.102,E2 27114.102} C_VEL
LIN {X 0,Y 561.369,Z 910.739,A -85,B 0,C 180,E1 27112.154,E2 27112.154} C_VEL
LIN {X 0,Y 560.91,Z 926.06,A -85,B 0,C 180,E1 27110.011,E2 27110.011} C_VEL
LIN {X 0,Y 560.563,Z 938.756,A -85,B 0,C 180,E1 27107.971,E2 27107.971} C_VEL
LIN {X 0,Y 560.3,Z 950.11,A -85,B 0,C 180,E1 27105.842,E2 27105.842} C_VEL
LIN {X 0,Y 560.13,Z 959.809,A -85,B 0,C 180,E1 27103.732,E2 27103.732} C_VEL
LIN {X 0,Y 560.015,Z 968.57,A -85,B 0,C 180,E1 27101.423,E2 27101.423} C_VEL
LIN {X 0,Y 559.95,Z 975.347,A -85,B 0,C 180,E1 27099.246,E2 27099.246} C_VEL
LIN {X 0,Y 559.898,Z 980.753,A -85,B 0,C 180,E1 27096.974,E2 27096.974} C_VEL
LIN {X 0,Y 559.909,Z 984.367,A -85,B 0,C 180,E1 27094.916,E2 27094.916} C_VEL
LIN {X 0,Y 559.913,Z 987.026,A -85,B 0,C 180,E1 27092.456,E2 27092.456} C_VEL
LIN {X 0,Y 559.894,Z 987.93,A -85,B 0,C 180,E1 27090.307,E2 27090.307} C_VEL
LIN {X 0,Y 559.914,Z 987.353,A -85,B 0,C 180,E1 27087.953,E2 27087.953} C_VEL
LIN {X 0,Y 559.913,Z 985.44,A -85,B 0,C 180,E1 27085.802,E2 27085.802} C_VEL
LIN {X 0,Y 559.916,Z 981.552,A -85,B 0,C 180,E1 27083.335,E2 27083.335} C_VEL
LIN {X 0,Y 559.944,Z 976.919,A -85,B 0,C 180,E1 27081.271,E2 27081.271} C_VEL
LIN {X 0,Y 559.984,Z 969.922,A -85,B 0,C 180,E1 27078.883,E2 27078.883} C_VEL
LIN {X 0,Y 560.096,Z 962.698,A -85,B 0,C 180,E1 27076.898,E2 27076.898} C_VEL
LIN {X 0,Y 560.271,Z 952.289,A -85,B 0,C 180,E1 27074.511,E2 27074.511} C_VEL
LIN {X 0,Y 560.501,Z 941.653,A -85,B 0,C 180,E1 27072.456,E2 27072.456} C_VEL
LIN {X 0,Y 560.845,Z 928.061,A -85,B 0,C 180,E1 27070.203,E2 27070.203} C_VEL
LIN {X 0,Y 561.281,Z 913.722,A -85,B 0,C 180,E1 27068.141,E2 27068.141} C_VEL
LIN {X 0,Y 561.81,Z 897.864,A -85,B 0,C 180,E1 27066.173,E2 27066.173} C_VEL
LIN {X 0,Y 562.435,Z 880.152,A -85,B 0,C 180,E1 27064.252,E2 27064.252} C_VEL
LIN {X 0,Y 563.097,Z 862.818,A -85,B 0,C 180,E1 27062.601,E2 27062.601} C_VEL
LIN {X 0,Y 563.819,Z 843.949,A -85,B 0,C 180,E1 27061.048,E2 27061.048} C_VEL
LIN {X 0,Y 564.582,Z 823.341,A -85,B 0,C 180,E1 27059.573,E2 27059.573} C_VEL
LIN {X 0,Y 565.322,Z 803.655,A -85,B 0,C 180,E1 27058.375,E2 27058.375} C_VEL
LIN {X 0,Y 566.044,Z 781.276,A -85,B 0,C 180,E1 27057.225,E2 27057.225} C_VEL
LIN {X 0,Y 566.686,Z 760.706,A -85,B 0,C 180,E1 27056.361,E2 27056.361} C_VEL
LIN {X 0,Y 567.256,Z 737.689,A -85,B 0,C 180,E1 27055.594,E2 27055.594} C_VEL
LIN {X 0,Y 567.672,Z 716.38,A -85,B 0,C 180,E1 27055.061,E2 27055.061} C_VEL
LIN {X 0,Y 568.033,Z 685.503,A -85,B 0,C 180,E1 27054.549,E2 27054.549} C_VEL
LIN {X 0,Y 569.479,Z 475.481,A -85,B 0,C 180,E1 27051.406,E2 27051.406} C_VEL
LIN {X 0,Y 570.039,Z 377.279,A -85,B 0,C 180,E1 27049.885,E2 27049.885} C_VEL
LIN {X 0,Y 565.19,Z 369.968,A -85,B 0,C 180,E1 27049.351,E2 27049.351} C_VEL
LIN {X 0,Y 562.751,Z 366.132,A -85,B 0,C 180,E1 27049.074,E2 27049.074} C_VEL
LIN {X 0,Y 560.731,Z 363.118,A -85,B 0,C 180,E1 27048.845,E2 27048.845} C_VEL
LIN {X 0,Y 560.276,Z 361.258,A -85,B 0,C 180,E1 27048.754,E2 27048.754} C_VEL
LIN {X 0,Y 560.258,Z 361.262,A -85,B 0,C 180,E1 27045.404,E2 27045.404} C_VEL
LIN {X 0,Y 560.277,Z 361.257,A -85,B 0,C 180,E1 27042.072,E2 27042.072} C_VEL
LIN {X 0,Y 560.246,Z 361.25,A -85,B 0,C 180,E1 27038.918,E2 27038.918} C_VEL
LIN {X 0,Y 560.275,Z 361.251,A -85,B 0,C 180,E1 27035.576,E2 27035.576} C_VEL
LIN {X 0,Y 560.266,Z 361.254,A -85,B 0,C 180,E1 27032.241,E2 27032.241} C_VEL
LIN {X 0,Y 560.239,Z 361.253,A -85,B 0,C 180,E1 27028.924,E2 27028.924} C_VEL
LIN {X 0,Y 560.283,Z 361.257,A -85,B 0,C 180,E1 27025.697,E2 27025.697} C_VEL
LIN {X 0,Y 560.228,Z 361.252,A -85,B 0,C 180,E1 27022.454,E2 27022.454} C_VEL
LIN {X 0,Y 560.271,Z 361.256,A -85,B 0,C 180,E1 27019.17,E2 27019.17} C_VEL
LIN {X 0,Y 560.236,Z 361.248,A -85,B 0,C 180,E1 27015.953,E2 27015.953} C_VEL
LIN {X 0,Y 560.225,Z 361.257,A -85,B 0,C 180,E1 27012.539,E2 27012.539} C_VEL
LIN {X 0,Y 560.273,Z 361.258,A -85,B 0,C 180,E1 27009.346,E2 27009.346} C_VEL
LIN {X 0,Y 560.211,Z 361.26,A -85,B 0,C 180,E1 27006.148,E2 27006.148} C_VEL
LIN {X 0,Y 560.276,Z 361.261,A -85,B 0,C 180,E1 27002.967,E2 27002.967} C_VEL
LIN {X 0,Y 560.204,Z 361.26,A -85,B 0,C 180,E1 26999.796,E2 26999.796} C_VEL
LIN {X 0,Y 560.239,Z 361.262,A -85,B 0,C 180,E1 26996.521,E2 26996.521} C_VEL
LIN {X 0,Y 560.198,Z 361.258,A -85,B 0,C 180,E1 26993.544,E2 26993.544} C_VEL
LIN {X 0,Y 560.22,Z 361.261,A -85,B 0,C 180,E1 26990.238,E2 26990.238} C_VEL
LIN {X 0,Y 560.203,Z 361.26,A -85,B 0,C 180,E1 26987.319,E2 26987.319} C_VEL
LIN {X 0,Y 560.217,Z 361.256,A -85,B 0,C 180,E1 26983.941,E2 26983.941} C_VEL
LIN {X 0,Y 560.226,Z 361.254,A -85,B 0,C 180,E1 26980.937,E2 26980.937} C_VEL
LIN {X 0,Y 560.214,Z 361.256,A -85,B 0,C 180,E1 26977.58,E2 26977.58} C_VEL
LIN {X 0,Y 560.275,Z 361.257,A -85,B 0,C 180,E1 26974.414,E2 26974.414} C_VEL
LIN {X 0,Y 560.216,Z 361.252,A -85,B 0,C 180,E1 26971.191,E2 26971.191} C_VEL
LIN {X 0,Y 560.282,Z 361.255,A -85,B 0,C 180,E1 26967.994,E2 26967.994} C_VEL
LIN {X 0,Y 560.227,Z 361.256,A -85,B 0,C 180,E1 26964.798,E2 26964.798} C_VEL
LIN {X 0,Y 560.248,Z 361.252,A -85,B 0,C 180,E1 26961.407,E2 26961.407} C_VEL
LIN {X 0,Y 560.262,Z 361.252,A -85,B 0,C 180,E1 26958.236,E2 26958.236} C_VEL
LIN {X 0,Y 560.236,Z 361.26,A -85,B 0,C 180,E1 26954.885,E2 26954.885} C_VEL
LIN {X 0,Y 560.308,Z 361.463,A -85,B 0,C 180,E1 26953.459,E2 26953.459} C_VEL
LIN {X 0,Y 561.46,Z 364.598,A -85,B 0,C 180,E1 26953.103,E2 26953.103} C_VEL
LIN {X 0,Y 567.619,Z 377.715,A -85,B 0,C 180,E1 26951.528,E2 26951.528} C_VEL
LIN {X 0,Y 568.269,Z 379.451,A -85,B 0,C 180,E1 26951.34,E2 26951.34} C_VEL
LIN {X 0,Y 568.061,Z 391.544,A -85,B 0,C 180,E1 26950.494,E2 26950.494} C_VEL
LIN {X 0,Y 570.262,Z 402.593,A -85,B 0,C 180,E1 26950.127,E2 26950.127} C_VEL
LIN {X 0,Y 568.71,Z 614.702,A -85,B 0,C 180,E1 26946.902,E2 26946.902} C_VEL
LIN {X 0,Y 567.808,Z 740.015,A -85,B 0,C 180,E1 26945.018,E2 26945.018} C_VEL
LIN {X 0,Y 567.322,Z 763.769,A -85,B 0,C 180,E1 26944.472,E2 26944.472} C_VEL
LIN {X 0,Y 566.85,Z 785.685,A -85,B 0,C 180,E1 26943.782,E2 26943.782} C_VEL
LIN {X 0,Y 566.161,Z 807.771,A -85,B 0,C 180,E1 26942.888,E2 26942.888} C_VEL
LIN {X 0,Y 565.504,Z 828.857,A -85,B 0,C 180,E1 26941.851,E2 26941.851} C_VEL
LIN {X 0,Y 564.72,Z 849.902,A -85,B 0,C 180,E1 26940.602,E2 26940.602} C_VEL
LIN {X 0,Y 563.957,Z 870.449,A -85,B 0,C 180,E1 26939.177,E2 26939.177} C_VEL
LIN {X 0,Y 563.249,Z 888.625,A -85,B 0,C 180,E1 26937.713,E2 26937.713} C_VEL
LIN {X 0,Y 562.525,Z 907.958,A -85,B 0,C 180,E1 26935.923,E2 26935.923} C_VEL
LIN {X 0,Y 561.904,Z 925.171,A -85,B 0,C 180,E1 26934.1,E2 26934.1} C_VEL
LIN {X 0,Y 561.358,Z 941.1,A -85,B 0,C 180,E1 26932.152,E2 26932.152} C_VEL
LIN {X 0,Y 560.901,Z 956.35,A -85,B 0,C 180,E1 26930.012,E2 26930.012} C_VEL
LIN {X 0,Y 560.561,Z 969.018,A -85,B 0,C 180,E1 26927.972,E2 26927.972} C_VEL
LIN {X 0,Y 560.297,Z 980.326,A -85,B 0,C 180,E1 26925.843,E2 26925.843} C_VEL
LIN {X 0,Y 560.127,Z 990.002,A -85,B 0,C 180,E1 26923.733,E2 26923.733} C_VEL
LIN {X 0,Y 560.021,Z 998.344,A -85,B 0,C 180,E1 26921.534,E2 26921.534} C_VEL
LIN {X 0,Y 559.944,Z 1004.871,A -85,B 0,C 180,E1 26919.455,E2 26919.455} C_VEL
LIN {X 0,Y 559.898,Z 1010.635,A -85,B 0,C 180,E1 26917.077,E2 26917.077} C_VEL
LIN {X 0,Y 559.91,Z 1014.277,A -85,B 0,C 180,E1 26915.02,E2 26915.02} C_VEL
LIN {X 0,Y 559.913,Z 1016.988,A -85,B 0,C 180,E1 26912.559,E2 26912.559} C_VEL
LIN {X 0,Y 559.887,Z 1017.917,A -85,B 0,C 180,E1 26910.41,E2 26910.41} C_VEL
LIN {X 0,Y 559.914,Z 1017.324,A -85,B 0,C 180,E1 26907.954,E2 26907.954} C_VEL
LIN {X 0,Y 559.908,Z 1015.277,A -85,B 0,C 180,E1 26905.699,E2 26905.699} C_VEL
LIN {X 0,Y 559.914,Z 1011.463,A -85,B 0,C 180,E1 26903.336,E2 26903.336} C_VEL
LIN {X 0,Y 559.946,Z 1006.809,A -85,B 0,C 180,E1 26901.271,E2 26901.271} C_VEL
LIN {X 0,Y 559.988,Z 999.77,A -85,B 0,C 180,E1 26898.883,E2 26898.883} C_VEL
LIN {X 0,Y 560.099,Z 992.116,A -85,B 0,C 180,E1 26896.793,E2 26896.793} C_VEL
LIN {X 0,Y 560.275,Z 981.893,A -85,B 0,C 180,E1 26894.475,E2 26894.475} C_VEL
LIN {X 0,Y 560.528,Z 970.833,A -85,B 0,C 180,E1 26892.35,E2 26892.35} C_VEL
LIN {X 0,Y 560.856,Z 957.771,A -85,B 0,C 180,E1 26890.204,E2 26890.204} C_VEL
LIN {X 0,Y 561.289,Z 943.347,A -85,B 0,C 180,E1 26888.138,E2 26888.138} C_VEL
LIN {X 0,Y 561.806,Z 927.969,A -85,B 0,C 180,E1 26886.231,E2 26886.231} C_VEL
LIN {X 0,Y 562.436,Z 910.151,A -85,B 0,C 180,E1 26884.297,E2 26884.297} C_VEL
LIN {X 0,Y 563.119,Z 892.257,A -85,B 0,C 180,E1 26882.595,E2 26882.595} C_VEL
LIN {X 0,Y 563.842,Z 873.39,A -85,B 0,C 180,E1 26881.05,E2 26881.05} C_VEL
LIN {X 0,Y 564.606,Z 852.669,A -85,B 0,C 180,E1 26879.575,E2 26879.575} C_VEL
LIN {X 0,Y 565.351,Z 832.907,A -85,B 0,C 180,E1 26878.378,E2 26878.378} C_VEL
LIN {X 0,Y 566.072,Z 810.174,A -85,B 0,C 180,E1 26877.22,E2 26877.22} C_VEL
LIN {X 0,Y 566.757,Z 788.886,A -85,B 0,C 180,E1 26876.336,E2 26876.336} C_VEL
LIN {X 0,Y 567.28,Z 766.028,A -85,B 0,C 180,E1 26875.591,E2 26875.591} C_VEL
LIN {X 0,Y 567.773,Z 743.367,A -85,B 0,C 180,E1 26875.042,E2 26875.042} C_VEL
LIN {X 0,Y 568.137,Z 699.738,A -85,B 0,C 180,E1 26874.361,E2 26874.361} C_VEL
LIN {X 0,Y 569.611,Z 488.421,A -85,B 0,C 180,E1 26871.192,E2 26871.192} C_VEL
LIN {X 0,Y 570.083,Z 400.859,A -85,B 0,C 180,E1 26869.83,E2 26869.83} C_VEL
LIN {X 0,Y 567.937,Z 390.789,A -85,B 0,C 180,E1 26869.476,E2 26869.476} C_VEL
LIN {X 0,Y 568.224,Z 379.12,A -85,B 0,C 180,E1 26868.631,E2 26868.631} C_VEL
LIN {X 0,Y 561.935,Z 365.269,A -85,B 0,C 180,E1 26866.995,E2 26866.995} C_VEL
LIN {X 0,Y 560.359,Z 361.769,A -85,B 0,C 180,E1 26866.57,E2 26866.57} C_VEL
LIN {X 0,Y 560.281,Z 361.247,A -85,B 0,C 180,E1 26866.468,E2 26866.468} C_VEL
LIN {X 0,Y 560.234,Z 361.259,A -85,B 0,C 180,E1 26863.261,E2 26863.261} C_VEL
LIN {X 0,Y 560.279,Z 361.26,A -85,B 0,C 180,E1 26859.974,E2 26859.974} C_VEL
LIN {X 0,Y 560.235,Z 361.259,A -85,B 0,C 180,E1 26856.751,E2 26856.751} C_VEL
LIN {X 0,Y 560.238,Z 361.259,A -85,B 0,C 180,E1 26853.345,E2 26853.345} C_VEL
LIN {X 0,Y 560.256,Z 361.255,A -85,B 0,C 180,E1 26850.216,E2 26850.216} C_VEL
LIN {X 0,Y 560.219,Z 361.26,A -85,B 0,C 180,E1 26846.957,E2 26846.957} C_VEL
LIN {X 0,Y 560.281,Z 361.245,A -85,B 0,C 180,E1 26843.741,E2 26843.741} C_VEL
LIN {X 0,Y 560.208,Z 361.26,A -85,B 0,C 180,E1 26840.585,E2 26840.585} C_VEL
LIN {X 0,Y 560.265,Z 361.247,A -85,B 0,C 180,E1 26837.339,E2 26837.339} C_VEL
LIN {X 0,Y 560.203,Z 361.261,A -85,B 0,C 180,E1 26834.259,E2 26834.259} C_VEL
LIN {X 0,Y 560.238,Z 361.262,A -85,B 0,C 180,E1 26831.009,E2 26831.009} C_VEL
LIN {X 0,Y 560.199,Z 361.261,A -85,B 0,C 180,E1 26828.002,E2 26828.002} C_VEL
LIN {X 0,Y 560.21,Z 361.262,A -85,B 0,C 180,E1 26824.606,E2 26824.606} C_VEL
LIN {X 0,Y 560.214,Z 361.259,A -85,B 0,C 180,E1 26821.636,E2 26821.636} C_VEL
LIN {X 0,Y 560.207,Z 361.258,A -85,B 0,C 180,E1 26818.261,E2 26818.261} C_VEL
LIN {X 0,Y 560.251,Z 361.262,A -85,B 0,C 180,E1 26815.188,E2 26815.188} C_VEL
LIN {X 0,Y 560.212,Z 361.259,A -85,B 0,C 180,E1 26811.997,E2 26811.997} C_VEL
LIN {X 0,Y 560.272,Z 361.261,A -85,B 0,C 180,E1 26808.887,E2 26808.887} C_VEL
LIN {X 0,Y 560.216,Z 361.26,A -85,B 0,C 180,E1 26805.7,E2 26805.7} C_VEL
LIN {X 0,Y 560.281,Z 361.244,A -85,B 0,C 180,E1 26802.554,E2 26802.554} C_VEL
